LIN {X 0,Y 681.209,Z 845.598,A -85,B 0,C 180,E1 31195.432,E2 31195.432} C_VEL
LIN {X 0,Y 674.082,Z 835.285,A -85,B 0,C 180,E1 31194.524,E2 31194.524} C_VEL
LIN {X 0,Y 668.532,Z 823.271,A -85,B 0,C 180,E1 31193.574,E2 31193.574} C_VEL
LIN {X 0,Y 664.818,Z 810.324,A -85,B 0,C 180,E1 31192.643,E2 31192.643} C_VEL
LIN {X 0,Y 662.53,Z 795.041,A -85,B 0,C 180,E1 31191.638,E2 31191.638} C_VEL
LIN {X 0,Y 661.762,Z 774.741,A -85,B 0,C 180,E1 31190.407,E2 31190.407} C_VEL
LIN {X 0,Y 664.221,Z 717.539,A -85,B 0,C 180,E1 31187.123,E2 31187.123} C_VEL
LIN {X 0,Y 665.52,Z 689.484,A -85,B 0,C 180,E1 31185.472,E2 31185.472} C_VEL
LIN {X 0,Y 655.199,Z 666.535,A -85,B 0,C 180,E1 31183.253,E2 31183.253} C_VEL
LIN {X 0,Y 648.915,Z 652.729,A -85,B 0,C 180,E1 31181.851,E2 31181.851} C_VEL
LIN {X 0,Y 648.754,Z 651.857,A -85,B 0,C 180,E1 31181.745,E2 31181.745} C_VEL
LIN {X 0,Y 648.762,Z 651.857,A -85,B 0,C 180,E1 31178.737,E2 31178.737} C_VEL
LIN {X 0,Y 648.769,Z 651.859,A -85,B 0,C 180,E1 31175.632,E2 31175.632} C_VEL
LIN {X 0,Y 648.783,Z 651.97,A -85,B 0,C 180,E1 31174.365,E2 31174.365} C_VEL
LIN {X 0,Y 654.485,Z 669.215,A -85,B 0,C 180,E1 31172.597,E2 31172.597} C_VEL
LIN {X 0,Y 656.821,Z 678.025,A -85,B 0,C 180,E1 31171.733,E2 31171.733} C_VEL
LIN {X 0,Y 656.243,Z 704.05,A -85,B 0,C 180,E1 31169.628,E2 31169.628} C_VEL
LIN {X 0,Y 659.956,Z 721.319,A -85,B 0,C 180,E1 31169.192,E2 31169.192} C_VEL
LIN {X 0,Y 658.097,Z 857.869,A -85,B 0,C 180,E1 31167.489,E2 31167.489} C_VEL
LIN {X 0,Y 656.788,Z 1005.042,A -85,B 0,C 180,E1 31165.748,E2 31165.748} C_VEL
LIN {X 0,Y 656.311,Z 1027.671,A -85,B 0,C 180,E1 31165.323,E2 31165.323} C_VEL
LIN {X 0,Y 655.768,Z 1048.897,A -85,B 0,C 180,E1 31164.769,E2 31164.769} C_VEL
LIN {X 0,Y 655.075,Z 1069.242,A -85,B 0,C 180,E1 31164.083,E2 31164.083} C_VEL
LIN {X 0,Y 654.302,Z 1088.647,A -85,B 0,C 180,E1 31163.268,E2 31163.268} C_VEL
LIN {X 0,Y 653.458,Z 1107.862,A -85,B 0,C 180,E1 31162.301,E2 31162.301} C_VEL
LIN {X 0,Y 652.558,Z 1127.004,A -85,B 0,C 180,E1 31161.152,E2 31161.152} C_VEL
LIN {X 0,Y 651.651,Z 1144.284,A -85,B 0,C 180,E1 31159.916,E2 31159.916} C_VEL
LIN {X 0,Y 650.775,Z 1161.184,A -85,B 0,C 180,E1 31158.499,E2 31158.499} C_VEL
LIN {X 0,Y 650.021,Z 1176.622,A -85,B 0,C 180,E1 31156.994,E2 31156.994} C_VEL
LIN {X 0,Y 649.364,Z 1190.989,A -85,B 0,C 180,E1 31155.358,E2 31155.358} C_VEL
LIN {X 0,Y 648.862,Z 1203.128,A -85,B 0,C 180,E1 31153.728,E2 31153.728} C_VEL
LIN {X 0,Y 648.463,Z 1214.556,A -85,B 0,C 180,E1 31151.924,E2 31151.924} C_VEL
LIN {X 0,Y 648.22,Z 1224.064,A -85,B 0,C 180,E1 31150.128,E2 31150.128} C_VEL
LIN {X 0,Y 648.047,Z 1232.048,A -85,B 0,C 180,E1 31148.25,E2 31148.25} C_VEL
LIN {X 0,Y 647.962,Z 1238.272,A -85,B 0,C 180,E1 31146.379,E2 31146.379} C_VEL
LIN {X 0,Y 647.927,Z 1242.932,A -85,B 0,C 180,E1 31144.498,E2 31144.498} C_VEL
LIN {X 0,Y 647.909,Z 1245.952,A -85,B 0,C 180,E1 31142.565,E2 31142.565} C_VEL
LIN {X 0,Y 647.912,Z 1247.338,A -85,B 0,C 180,E1 31140.619,E2 31140.619} C_VEL
LIN {X 0,Y 647.903,Z 1247.184,A -85,B 0,C 180,E1 31138.762,E2 31138.762} C_VEL
LIN {X 0,Y 647.901,Z 1245.342,A -85,B 0,C 180,E1 31136.865,E2 31136.865} C_VEL
LIN {X 0,Y 647.927,Z 1241.709,A -85,B 0,C 180,E1 31134.865,E2 31134.865} C_VEL
LIN {X 0,Y 647.985,Z 1236.727,A -85,B 0,C 180,E1 31132.998,E2 31132.998} C_VEL
LIN {X 0,Y 648.081,Z 1229.943,A -85,B 0,C 180,E1 31131.125,E2 31131.125} C_VEL
LIN {X 0,Y 648.276,Z 1221.361,A -85,B 0,C 180,E1 31129.244,E2 31129.244} C_VEL
LIN {X 0,Y 648.58,Z 1211.375,A -85,B 0,C 180,E1 31127.445,E2 31127.445} C_VEL
LIN {X 0,Y 648.998,Z 1199.871,A -85,B 0,C 180,E1 31125.716,E2 31125.716} C_VEL
LIN {X 0,Y 649.525,Z 1187.153,A -85,B 0,C 180,E1 31124.096,E2 31124.096} C_VEL
LIN {X 0,Y 650.223,Z 1172.154,A -85,B 0,C 180,E1 31122.458,E2 31122.458} C_VEL
LIN {X 0,Y 651.031,Z 1156.602,A -85,B 0,C 180,E1 31120.998,E2 31120.998} C_VEL
LIN {X 0,Y 651.882,Z 1140.018,A -85,B 0,C 180,E1 31119.67,E2 31119.67} C_VEL
LIN {X 0,Y 652.795,Z 1121.9,A -85,B 0,C 180,E1 31118.432,E2 31118.432} C_VEL
LIN {X 0,Y 653.743,Z 1102.903,A -85,B 0,C 180,E1 31117.329,E2 31117.329} C_VEL
LIN {X 0,Y 654.621,Z 1083.016,A -85,B 0,C 180,E1 31116.362,E2 31116.362} C_VEL
LIN {X 0,Y 655.426,Z 1063.233,A -85,B 0,C 180,E1 31115.58,E2 31115.58} C_VEL
LIN {X 0,Y 656.167,Z 1040.826,A -85,B 0,C 180,E1 31114.87,E2 31114.87} C_VEL
LIN {X 0,Y 656.776,Z 1019.125,A -85,B 0,C 180,E1 31114.351,E2 31114.351} C_VEL
LIN {X 0,Y 657.189,Z 997.108,A -85,B 0,C 180,E1 31113.988,E2 31113.988} C_VEL
LIN {X 0,Y 657.978,Z 910.113,A -85,B 0,C 180,E1 31112.971,E2 31112.971} C_VEL
LIN {X 0,Y 657.137,Z 902.528,A -85,B 0,C 180,E1 31112.844,E2 31112.844} C_VEL
LIN {X 0,Y 651.672,Z 882.715,A -85,B 0,C 180,E1 31112.37,E2 31112.37} C_VEL
LIN {X 0,Y 651.081,Z 876.194,A -85,B 0,C 180,E1 31112.264,E2 31112.264} C_VEL
LIN {X 0,Y 652.864,Z 721.354,A -85,B 0,C 180,E1 31110.361,E2 31110.361} C_VEL
LIN {X 0,Y 648.381,Z 701.444,A -85,B 0,C 180,E1 31109.856,E2 31109.856} C_VEL
LIN {X 0,Y 649.101,Z 679.474,A -85,B 0,C 180,E1 31108.001,E2 31108.001} C_VEL
LIN {X 0,Y 642.45,Z 657.995,A -85,B 0,C 180,E1 31105.735,E2 31105.735} C_VEL
LIN {X 0,Y 640.828,Z 652.848,A -85,B 0,C 180,E1 31105.158,E2 31105.158} C_VEL
LIN {X 0,Y 640.828,Z 652.845,A -85,B 0,C 180,E1 31101.952,E2 31101.952} C_VEL
LIN {X 0,Y 640.831,Z 652.844,A -85,B 0,C 180,E1 31098.818,E2 31098.818} C_VEL
LIN {X 0,Y 640.829,Z 652.843,A -85,B 0,C 180,E1 31095.613,E2 31095.613} C_VEL
LIN {X 0,Y 640.819,Z 652.84,A -85,B 0,C 180,E1 31092.435,E2 31092.435} C_VEL
LIN {X 0,Y 640.82,Z 652.846,A -85,B 0,C 180,E1 31089.292,E2 31089.292} C_VEL
LIN {X 0,Y 640.831,Z 652.845,A -85,B 0,C 180,E1 31086.227,E2 31086.227} C_VEL
LIN {X 0,Y 640.827,Z 652.841,A -85,B 0,C 180,E1 31082.995,E2 31082.995} C_VEL
LIN {X 0,Y 640.816,Z 652.84,A -85,B 0,C 180,E1 31079.852,E2 31079.852} C_VEL
LIN {X 0,Y 640.82,Z 652.844,A -85,B 0,C 180,E1 31076.805,E2 31076.805} C_VEL
LIN {X 0,Y 640.831,Z 652.847,A -85,B 0,C 180,E1 31073.666,E2 31073.666} C_VEL
LIN {X 0,Y 640.827,Z 652.843,A -85,B 0,C 180,E1 31070.458,E2 31070.458} C_VEL
LIN {X 0,Y 640.815,Z 652.841,A -85,B 0,C 180,E1 31067.34,E2 31067.34} C_VEL
LIN {X 0,Y 640.816,Z 652.841,A -85,B 0,C 180,E1 31064.273,E2 31064.273} C_VEL
LIN {X 0,Y 640.829,Z 652.847,A -85,B 0,C 180,E1 31061.157,E2 31061.157} C_VEL
LIN {X 0,Y 640.827,Z 652.837,A -85,B 0,C 180,E1 31057.983,E2 31057.983} C_VEL
LIN {X 0,Y 640.817,Z 652.839,A -85,B 0,C 180,E1 31054.924,E2 31054.924} C_VEL
LIN {X 0,Y 640.816,Z 652.843,A -85,B 0,C 180,E1 31051.789,E2 31051.789} C_VEL
LIN {X 0,Y 640.832,Z 652.844,A -85,B 0,C 180,E1 31048.75,E2 31048.75} C_VEL
LIN {X 0,Y 640.828,Z 652.839,A -85,B 0,C 180,E1 31045.527,E2 31045.527} C_VEL
LIN {X 0,Y 640.816,Z 652.838,A -85,B 0,C 180,E1 31042.47,E2 31042.47} C_VEL
LIN {X 0,Y 640.82,Z 652.84,A -85,B 0,C 180,E1 31039.392,E2 31039.392} C_VEL
LIN {X 0,Y 640.832,Z 652.846,A -85,B 0,C 180,E1 31036.282,E2 31036.282} C_VEL
LIN {X 0,Y 640.83,Z 652.842,A -85,B 0,C 180,E1 31033.131,E2 31033.131} C_VEL
LIN {X 0,Y 640.82,Z 652.839,A -85,B 0,C 180,E1 31030.02,E2 31030.02} C_VEL
LIN {X 0,Y 640.824,Z 652.844,A -85,B 0,C 180,E1 31026.945,E2 31026.945} C_VEL
LIN {X 0,Y 640.833,Z 652.847,A -85,B 0,C 180,E1 31023.789,E2 31023.789} C_VEL
LIN {X 0,Y 640.831,Z 652.842,A -85,B 0,C 180,E1 31020.666,E2 31020.666} C_VEL
LIN {X 0,Y 640.82,Z 652.834,A -85,B 0,C 180,E1 31017.539,E2 31017.539} C_VEL
LIN {X 0,Y 640.819,Z 652.838,A -85,B 0,C 180,E1 31014.384,E2 31014.384} C_VEL
LIN {X 0,Y 640.836,Z 652.84,A -85,B 0,C 180,E1 31011.27,E2 31011.27} C_VEL
LIN {X 0,Y 640.829,Z 652.839,A -85,B 0,C 180,E1 31008.097,E2 31008.097} C_VEL
LIN {X 0,Y 640.817,Z 652.846,A -85,B 0,C 180,E1 31004.978,E2 31004.978} C_VEL
LIN {X 0,Y 640.82,Z 652.884,A -85,B 0,C 180,E1 31003.553,E2 31003.553} C_VEL
LIN {X 0,Y 650.521,Z 680.608,A -85,B 0,C 180,E1 31000.787,E2 31000.787} C_VEL
LIN {X 0,Y 651.272,Z 683.79,A -85,B 0,C 180,E1 31000.499,E2 31000.499} C_VEL
LIN {X 0,Y 649.818,Z 722.359,A -85,B 0,C 180,E1 30997.653,E2 30997.653} C_VEL
LIN {X 0,Y 648.069,Z 765.963,A -85,B 0,C 180,E1 30994.488,E2 30994.488} C_VEL
LIN {X 0,Y 646.393,Z 811.774,A -85,B 0,C 180,E1 30991.212,E2 30991.212} C_VEL
LIN {X 0,Y 644.846,Z 859.861,A -85,B 0,C 180,E1 30987.822,E2 30987.822} C_VEL
LIN {X 0,Y 643.902,Z 897.134,A -85,B 0,C 180,E1 30985.254,E2 30985.254} C_VEL
LIN {X 0,Y 644.559,Z 904.252,A -85,B 0,C 180,E1 30985.14,E2 30985.14} C_VEL
LIN {X 0,Y 643.103,Z 1040.339,A -85,B 0,C 180,E1 30983.376,E2 30983.376} C_VEL
LIN {X 0,Y 642.901,Z 1057.395,A -85,B 0,C 180,E1 30982.978,E2 30982.978} C_VEL
LIN {X 0,Y 642.615,Z 1072.675,A -85,B 0,C 180,E1 30982.451,E2 30982.451} C_VEL
LIN {X 0,Y 642.248,Z 1087.818,A -85,B 0,C 180,E1 30981.749,E2 30981.749} C_VEL
LIN {X 0,Y 641.886,Z 1101.299,A -85,B 0,C 180,E1 30980.947,E2 30980.947} C_VEL
LIN {X 0,Y 641.498,Z 1114.46,A -85,B 0,C 180,E1 30979.959,E2 30979.959} C_VEL
LIN {X 0,Y 641.17,Z 1125.58,A -85,B 0,C 180,E1 30978.928,E2 30978.928} C_VEL
LIN {X 0,Y 640.845,Z 1136.028,A -85,B 0,C 180,E1 30977.713,E2 30977.713} C_VEL
LIN {X 0,Y 640.602,Z 1144.93,A -85,B 0,C 180,E1 30976.411,E2 30976.411} C_VEL
LIN {X 0,Y 640.42,Z 1152.141,A -85,B 0,C 180,E1 30975.021,E2 30975.021} C_VEL
LIN {X 0,Y 640.328,Z 1157.431,A -85,B 0,C 180,E1 30973.638,E2 30973.638} C_VEL
LIN {X 0,Y 640.278,Z 1161.119,A -85,B 0,C 180,E1 30972.162,E2 30972.162} C_VEL
LIN {X 0,Y 640.258,Z 1163.071,A -85,B 0,C 180,E1 30970.619,E2 30970.619} C_VEL
LIN {X 0,Y 640.272,Z 1163.08,A -85,B 0,C 180,E1 30969.166,E2 30969.166} C_VEL
LIN {X 0,Y 640.325,Z 1161.258,A -85,B 0,C 180,E1 30967.627,E2 30967.627} C_VEL
LIN {X 0,Y 640.398,Z 1157.705,A -85,B 0,C 180,E1 30966.185,E2 30966.185} C_VEL
LIN {X 0,Y 640.541,Z 1152.319,A -85,B 0,C 180,E1 30964.746,E2 30964.746} C_VEL
LIN {X 0,Y 640.756,Z 1145.362,A -85,B 0,C 180,E1 30963.4,E2 30963.4} C_VEL
LIN {X 0,Y 641.066,Z 1136.322,A -85,B 0,C 180,E1 30962.056,E2 30962.056} C_VEL
LIN {X 0,Y 641.419,Z 1126.338,A -85,B 0,C 180,E1 30960.893,E2 30960.893} C_VEL
LIN {X 0,Y 641.835,Z 1114.407,A -85,B 0,C 180,E1 30959.777,E2 30959.777} C_VEL
LIN {X 0,Y 642.239,Z 1101.835,A -85,B 0,C 180,E1 30958.84,E2 30958.84} C_VEL
LIN {X 0,Y 642.653,Z 1087.565,A -85,B 0,C 180,E1 30957.994,E2 30957.994} C_VEL
LIN {X 0,Y 643.023,Z 1072.906,A -85,B 0,C 180,E1 30957.326,E2 30957.326} C_VEL
LIN {X 0,Y 643.302,Z 1057.109,A -85,B 0,C 180,E1 30956.792,E2 30956.792} C_VEL
LIN {X 0,Y 643.467,Z 1041.097,A -85,B 0,C 180,E1 30956.428,E2 30956.428} C_VEL
LIN {X 0,Y 645.88,Z 902.439,A -85,B 0,C 180,E1 30954.392,E2 30954.392} C_VEL
LIN {X 0,Y 648,Z 858.527,A -85,B 0,C 180,E1 30951.168,E2 30951.168} C_VEL
LIN {X 0,Y 650.67,Z 813.787,A -85,B 0,C 180,E1 30947.802,E2 30947.802} C_VEL
LIN {X 0,Y 653.996,Z 769.687,A -85,B 0,C 180,E1 30944.39,E2 30944.39} C_VEL
LIN {X 0,Y 657.874,Z 728.174,A -85,B 0,C 180,E1 30941.065,E2 30941.065} C_VEL
LIN {X 0,Y 660.552,Z 697.265,A -85,B 0,C 180,E1 30938.418,E2 30938.418} C_VEL
LIN {X 0,Y 655.76,Z 684.811,A -85,B 0,C 180,E1 30936.618,E2 30936.618} C_VEL
LIN {X 0,Y 651.47,Z 674.698,A -85,B 0,C 180,E1 30934.937,E2 30934.937} C_VEL
LIN {X 0,Y 647.844,Z 666.788,A -85,B 0,C 180,E1 30933.411,E2 30933.411} C_VEL
LIN {X 0,Y 646.119,Z 663.273,A -85,B 0,C 180,E1 30932.637,E2 30932.637} C_VEL
LIN {X 0,Y 643.776,Z 658.862,A -85,B 0,C 180,E1 30931.522,E2 30931.522} C_VEL
LIN {X 0,Y 643.304,Z 657.701,A -85,B 0,C 180,E1 30931.234,E2 30931.234} C_VEL
LIN {X 0,Y 641.165,Z 654.377,A -85,B 0,C 180,E1 30930.117,E2 30930.117} C_VEL
LIN {X 0,Y 640.815,Z 652.847,A -85,B 0,C 180,E1 30929.632,E2 30929.632} C_VEL
LIN {X 0,Y 640.817,Z 652.848,A -85,B 0,C 180,E1 30926.578,E2 30926.578} C_VEL
LIN {X 0,Y 640.814,Z 652.848,A -85,B 0,C 180,E1 30923.47,E2 30923.47} C_VEL
LIN {X 0,Y 640.847,Z 652.979,A -85,B 0,C 180,E1 30921.097,E2 30921.097} C_VEL
LIN {X 0,Y 642.181,Z 656.406,A -85,B 0,C 180,E1 30920.213,E2 30920.213} C_VEL
LIN {X 0,Y 643.755,Z 658.201,A -85,B 0,C 180,E1 30919.632,E2 30919.632} C_VEL
LIN {X 0,Y 645.497,Z 662.058,A -85,B 0,C 180,E1 30918.827,E2 30918.827} C_VEL
LIN {X 0,Y 646.606,Z 663.902,A -85,B 0,C 180,E1 30918.441,E2 30918.441} C_VEL
LIN {X 0,Y 649.083,Z 668.897,A -85,B 0,C 180,E1 30917.549,E2 30917.549} C_VEL
LIN {X 0,Y 652.65,Z 676.198,A -85,B 0,C 180,E1 30916.415,E2 30916.415} C_VEL
LIN {X 0,Y 657.722,Z 688.151,A -85,B 0,C 180,E1 30914.893,E2 30914.893} C_VEL
LIN {X 0,Y 658.832,Z 691.207,A -85,B 0,C 180,E1 30914.557,E2 30914.557} C_VEL
LIN {X 0,Y 654.691,Z 733.352,A -85,B 0,C 180,E1 30911.945,E2 30911.945} C_VEL
LIN {X 0,Y 652.167,Z 775.541,A -85,B 0,C 180,E1 30909.449,E2 30909.449} C_VEL
LIN {X 0,Y 653.059,Z 796.061,A -85,B 0,C 180,E1 30908.174,E2 30908.174} C_VEL
LIN {X 0,Y 655.531,Z 811.396,A -85,B 0,C 180,E1 30907.156,E2 30907.156} C_VEL
LIN {X 0,Y 659.426,Z 824.494,A -85,B 0,C 180,E1 30906.227,E2 30906.227} C_VEL
LIN {X 0,Y 665.197,Z 836.86,A -85,B 0,C 180,E1 30905.292,E2 30905.292} C_VEL
LIN {X 0,Y 672.623,Z 847.758,A -85,B 0,C 180,E1 30904.407,E2 30904.407} C_VEL
LIN {X 0,Y 681.659,Z 857.265,A -85,B 0,C 180,E1 30903.574,E2 30903.574} C_VEL
LIN {X 0,Y 691.482,Z 864.868,A -85,B 0,C 180,E1 30902.845,E2 30902.845} C_VEL
LIN {X 0,Y 702.753,Z 871.277,A -85,B 0,C 180,E1 30902.158,E2 30902.158} C_VEL
LIN {X 0,Y 715.436,Z 876.288,A -85,B 0,C 180,E1 30901.511,E2 30901.511} C_VEL
LIN {X 0,Y 720.879,Z 877.314,A -85,B 0,C 180,E1 30901.151,E2 30901.151} C_VEL
LIN {X 0,Y 724.061,Z 877.311,A -85,B 0,C 180,E1 30900.847,E2 30900.847} C_VEL
LIN {X 0,Y 720.157,Z 886.663,A -85,B 0,C 180,E1 30900.632,E2 30900.632} C_VEL
LIN {X 0,Y 710.62,Z 902.495,A -85,B 0,C 180,E1 30900.397,E2 30900.397} C_VEL
LIN {X 0,Y 697.384,Z 921.767,A -85,B 0,C 180,E1 30899.929,E2 30899.929} C_VEL
LIN {X 0,Y 679.73,Z 948.078,A -85,B 0,C 180,E1 30899.184,E2 30899.184} C_VEL
LIN {X 0,Y 670.449,Z 964.538,A -85,B 0,C 180,E1 30898.649,E2 30898.649} C_VEL
LIN {X 0,Y 664.344,Z 978.497,A -85,B 0,C 180,E1 30898.136,E2 30898.136} C_VEL
LIN {X 0,Y 662.043,Z 984.008,A -85,B 0,C 180,E1 30897.928,E2 30897.928} C_VEL
LIN {X 0,Y 656.266,Z 997.296,A -85,B 0,C 180,E1 30897.428,E2 30897.428} C_VEL
LIN {X 0,Y 650.15,Z 1017.526,A -85,B 0,C 180,E1 30896.584,E2 30896.584} C_VEL
LIN {X 0,Y 649.41,Z 1021.143,A -85,B 0,C 180,E1 30896.453,E2 30896.453} C_VEL
LIN {X 0,Y 648.837,Z 1062.962,A -85,B 0,C 180,E1 30895.95,E2 30895.95} C_VEL
LIN {X 0,Y 648.281,Z 1086.804,A -85,B 0,C 180,E1 30895.491,E2 30895.491} C_VEL
LIN {X 0,Y 647.655,Z 1109.654,A -85,B 0,C 180,E1 30894.877,E2 30894.877} C_VEL
LIN {X 0,Y 646.894,Z 1131.523,A -85,B 0,C 180,E1 30894.115,E2 30894.115} C_VEL
LIN {X 0,Y 646.063,Z 1153.311,A -85,B 0,C 180,E1 30893.173,E2 30893.173} C_VEL
LIN {X 0,Y 645.207,Z 1173.52,A -85,B 0,C 180,E1 30892.12,E2 30892.12} C_VEL
LIN {X 0,Y 644.365,Z 1192.384,A -85,B 0,C 180,E1 30890.956,E2 30890.956} C_VEL
LIN {X 0,Y 643.526,Z 1209.876,A -85,B 0,C 180,E1 30889.68,E2 30889.68} C_VEL
LIN {X 0,Y 642.771,Z 1226.068,A -85,B 0,C 180,E1 30888.313,E2 30888.313} C_VEL
LIN {X 0,Y 642.061,Z 1239.527,A -85,B 0,C 180,E1 30886.929,E2 30886.929} C_VEL
LIN {X 0,Y 641.481,Z 1251.253,A -85,B 0,C 180,E1 30885.55,E2 30885.55} C_VEL
LIN {X 0,Y 640.968,Z 1262.832,A -85,B 0,C 180,E1 30883.991,E2 30883.991} C_VEL
LIN {X 0,Y 640.52,Z 1274.803,A -85,B 0,C 180,E1 30882.073,E2 30882.073} C_VEL
LIN {X 0,Y 640.251,Z 1283.342,A -85,B 0,C 180,E1 30880.436,E2 30880.436} C_VEL
LIN {X 0,Y 640.081,Z 1290.854,A -85,B 0,C 180,E1 30878.714,E2 30878.714} C_VEL
LIN {X 0,Y 639.963,Z 1297.62,A -85,B 0,C 180,E1 30876.728,E2 30876.728} C_VEL
LIN {X 0,Y 639.927,Z 1301.986,A -85,B 0,C 180,E1 30875.019,E2 30875.019} C_VEL
LIN {X 0,Y 639.919,Z 1305.213,A -85,B 0,C 180,E1 30873.223,E2 30873.223} C_VEL
LIN {X 0,Y 639.914,Z 1307.192,A -85,B 0,C 180,E1 30871.073,E2 30871.073} C_VEL
LIN {X 0,Y 639.904,Z 1307.328,A -85,B 0,C 180,E1 30869.372,E2 30869.372} C_VEL
LIN {X 0,Y 639.905,Z 1306.259,A -85,B 0,C 180,E1 30867.67,E2 30867.67} C_VEL
LIN {X 0,Y 639.923,Z 1303.51,A -85,B 0,C 180,E1 30865.698,E2 30865.698} C_VEL
LIN {X 0,Y 639.952,Z 1299.128,A -85,B 0,C 180,E1 30863.81,E2 30863.81} C_VEL
LIN {X 0,Y 640.019,Z 1294.119,A -85,B 0,C 180,E1 30862.187,E2 30862.187} C_VEL
LIN {X 0,Y 640.162,Z 1287.481,A -85,B 0,C 180,E1 30860.469,E2 30860.469} C_VEL
LIN {X 0,Y 640.42,Z 1277.822,A -85,B 0,C 180,E1 30858.471,E2 30858.471} C_VEL
LIN {X 0,Y 640.728,Z 1268.768,A -85,B 0,C 180,E1 30856.921,E2 30856.921} C_VEL
LIN {X 0,Y 641.138,Z 1258.901,A -85,B 0,C 180,E1 30855.457,E2 30855.457} C_VEL
LIN {X 0,Y 641.747,Z 1246.072,A -85,B 0,C 180,E1 30853.805,E2 30853.805} C_VEL
LIN {X 0,Y 642.465,Z 1231.649,A -85,B 0,C 180,E1 30852.238,E2 30852.238} C_VEL
LIN {X 0,Y 643.038,Z 1220.295,A -85,B 0,C 180,E1 30851.176,E2 30851.176} C_VEL
LIN {X 0,Y 643.729,Z 1206.008,A -85,B 0,C 180,E1 30850.008,E2 30850.008} C_VEL
LIN {X 0,Y 644.577,Z 1189.105,A -85,B 0,C 180,E1 30848.796,E2 30848.796} C_VEL
LIN {X 0,Y 645.498,Z 1169.439,A -85,B 0,C 180,E1 30847.6,E2 30847.6} C_VEL
LIN {X 0,Y 646.44,Z 1148.388,A -85,B 0,C 180,E1 30846.525,E2 30846.525} C_VEL
LIN {X 0,Y 647.307,Z 1127.423,A -85,B 0,C 180,E1 30845.641,E2 30845.641} C_VEL
LIN {X 0,Y 648.102,Z 1105.683,A -85,B 0,C 180,E1 30844.908,E2 30844.908} C_VEL
LIN {X 0,Y 648.775,Z 1083.009,A -85,B 0,C 180,E1 30844.321,E2 30844.321} C_VEL
LIN {X 0,Y 649.317,Z 1060.66,A -85,B 0,C 180,E1 30843.904,E2 30843.904} C_VEL
LIN {X 0,Y 649.898,Z 1021.34,A -85,B 0,C 180,E1 30843.427,E2 30843.427} C_VEL
LIN {X 0,Y 653.512,Z 1008.382,A -85,B 0,C 180,E1 30842.873,E2 30842.873} C_VEL
LIN {X 0,Y 658.239,Z 994.241,A -85,B 0,C 180,E1 30842.3,E2 30842.3} C_VEL
LIN {X 0,Y 664.396,Z 980.423,A -85,B 0,C 180,E1 30841.799,E2 30841.799} C_VEL
LIN {X 0,Y 669.874,Z 967.309,A -85,B 0,C 180,E1 30841.321,E2 30841.321} C_VEL
LIN {X 0,Y 678.652,Z 950.97,A -85,B 0,C 180,E1 30840.811,E2 30840.811} C_VEL
LIN {X 0,Y 693.309,Z 928.11,A -85,B 0,C 180,E1 30840.203,E2 30840.203} C_VEL
LIN {X 0,Y 712.087,Z 900.21,A -85,B 0,C 180,E1 30839.561,E2 30839.561} C_VEL
LIN {X 0,Y 720.725,Z 885.47,A -85,B 0,C 180,E1 30839.346,E2 30839.346} C_VEL
LIN {X 0,Y 724.073,Z 877.281,A -85,B 0,C 180,E1 30839.152,E2 30839.152} C_VEL
LIN {X 0,Y 719.403,Z 877.155,A -85,B 0,C 180,E1 30838.736,E2 30838.736} C_VEL
LIN {X 0,Y 713.768,Z 875.787,A -85,B 0,C 180,E1 30838.4,E2 30838.4} C_VEL
LIN {X 0,Y 701.67,Z 871.121,A -85,B 0,C 180,E1 30837.676,E2 30837.676} C_VEL
LIN {X 0,Y 691.019,Z 865.082,A -85,B 0,C 180,E1 30836.909,E2 30836.909} C_VEL
LIN {X 0,Y 681.773,Z 857.782,A -85,B 0,C 180,E1 30836.109,E2 30836.109} C_VEL
LIN {X 0,Y 673.653,Z 848.946,A -85,B 0,C 180,E1 30835.252,E2 30835.252} C_VEL
LIN {X 0,Y 666.592,Z 838.079,A -85,B 0,C 180,E1 30834.302,E2 30834.302} C_VEL
LIN {X 0,Y 661.173,Z 825.61,A -85,B 0,C 180,E1 30833.318,E2 30833.318} C_VEL
LIN {X 0,Y 657.433,Z 811.523,A -85,B 0,C 180,E1 30832.308,E2 30832.308} C_VEL
LIN {X 0,Y 655.376,Z 795.861,A -85,B 0,C 180,E1 30831.278,E2 30831.278} C_VEL
LIN {X 0,Y 654.815,Z 775.606,A -85,B 0,C 180,E1 30830.045,E2 30830.045} C_VEL
LIN {X 0,Y 657.442,Z 719.808,A -85,B 0,C 180,E1 30826.811,E2 30826.811} C_VEL
LIN {X 0,Y 658.829,Z 693.191,A -85,B 0,C 180,E1 30825.234,E2 30825.234} C_VEL
LIN {X 0,Y 647.655,Z 668.207,A -85,B 0,C 180,E1 30822.789,E2 30822.789} C_VEL
LIN {X 0,Y 641.688,Z 655.612,A -85,B 0,C 180,E1 30821.471,E2 30821.471} C_VEL
LIN {X 0,Y 640.829,Z 652.848,A -85,B 0,C 180,E1 30821.182,E2 30821.182} C_VEL
LIN {X 0,Y 640.832,Z 652.847,A -85,B 0,C 180,E1 30818.005,E2 30818.005} C_VEL
LIN {X 0,Y 640.861,Z 653.038,A -85,B 0,C 180,E1 30814.846,E2 30814.846} C_VEL
LIN {X 0,Y 646.617,Z 669.593,A -85,B 0,C 180,E1 30813.084,E2 30813.084} C_VEL
LIN {X 0,Y 649.738,Z 680.661,A -85,B 0,C 180,E1 30811.964,E2 30811.964} C_VEL
LIN {X 0,Y 649.191,Z 704.841,A -85,B 0,C 180,E1 30810.004,E2 30810.004} C_VEL
LIN {X 0,Y 653.002,Z 722.678,A -85,B 0,C 180,E1 30809.526,E2 30809.526} C_VEL
LIN {X 0,Y 650.797,Z 859.006,A -85,B 0,C 180,E1 30807.766,E2 30807.766} C_VEL
LIN {X 0,Y 649.316,Z 1005.981,A -85,B 0,C 180,E1 30805.99,E2 30805.99} C_VEL
LIN {X 0,Y 648.819,Z 1028.459,A -85,B 0,C 180,E1 30805.561,E2 30805.561} C_VEL
LIN {X 0,Y 648.22,Z 1050.332,A -85,B 0,C 180,E1 30804.978,E2 30804.978} C_VEL
LIN {X 0,Y 647.477,Z 1071.362,A -85,B 0,C 180,E1 30804.254,E2 30804.254} C_VEL
LIN {X 0,Y 646.61,Z 1091.799,A -85,B 0,C 180,E1 30803.368,E2 30803.368} C_VEL
LIN {X 0,Y 645.678,Z 1111.353,A -85,B 0,C 180,E1 30802.345,E2 30802.345} C_VEL
LIN {X 0,Y 644.8,Z 1128.969,A -85,B 0,C 180,E1 30801.255,E2 30801.255} C_VEL
LIN {X 0,Y 643.884,Z 1145.8,A -85,B 0,C 180,E1 30800.03,E2 30800.03} C_VEL
LIN {X 0,Y 643.019,Z 1161.653,A -85,B 0,C 180,E1 30798.683,E2 30798.683} C_VEL
LIN {X 0,Y 642.227,Z 1176.625,A -85,B 0,C 180,E1 30797.206,E2 30797.206} C_VEL
LIN {X 0,Y 641.508,Z 1190.991,A -85,B 0,C 180,E1 30795.551,E2 30795.551} C_VEL
LIN {X 0,Y 640.956,Z 1203.13,A -85,B 0,C 180,E1 30793.901,E2 30793.901} C_VEL
LIN {X 0,Y 640.52,Z 1214.557,A -85,B 0,C 180,E1 30792.074,E2 30792.074} C_VEL
LIN {X 0,Y 640.252,Z 1224.067,A -85,B 0,C 180,E1 30790.255,E2 30790.255} C_VEL
LIN {X 0,Y 640.056,Z 1232.05,A -85,B 0,C 180,E1 30788.354,E2 30788.354} C_VEL
LIN {X 0,Y 639.964,Z 1238.342,A -85,B 0,C 180,E1 30786.435,E2 30786.435} C_VEL
LIN {X 0,Y 639.927,Z 1242.984,A -85,B 0,C 180,E1 30784.525,E2 30784.525} C_VEL
LIN {X 0,Y 639.91,Z 1245.952,A -85,B 0,C 180,E1 30782.597,E2 30782.597} C_VEL
LIN {X 0,Y 639.912,Z 1247.338,A -85,B 0,C 180,E1 30780.627,E2 30780.627} C_VEL
LIN {X 0,Y 639.903,Z 1247.184,A -85,B 0,C 180,E1 30778.746,E2 30778.746} C_VEL
LIN {X 0,Y 639.901,Z 1245.367,A -85,B 0,C 180,E1 30776.847,E2 30776.847} C_VEL
LIN {X 0,Y 639.93,Z 1241.708,A -85,B 0,C 180,E1 30774.8,E2 30774.8} C_VEL
LIN {X 0,Y 639.993,Z 1236.725,A -85,B 0,C 180,E1 30772.91,E2 30772.91} C_VEL
LIN {X 0,Y 640.103,Z 1229.941,A -85,B 0,C 180,E1 30771.013,E2 30771.013} C_VEL
LIN {X 0,Y 640.317,Z 1221.357,A -85,B 0,C 180,E1 30769.109,E2 30769.109} C_VEL
LIN {X 0,Y 640.648,Z 1211.348,A -85,B 0,C 180,E1 30767.284,E2 30767.284} C_VEL
LIN {X 0,Y 641.103,Z 1199.957,A -85,B 0,C 180,E1 30765.549,E2 30765.549} C_VEL
LIN {X 0,Y 641.686,Z 1187.145,A -85,B 0,C 180,E1 30763.897,E2 30763.897} C_VEL
LIN {X 0,Y 642.445,Z 1172.146,A -85,B 0,C 180,E1 30762.239,E2 30762.239} C_VEL
LIN {X 0,Y 643.315,Z 1156.535,A -85,B 0,C 180,E1 30760.761,E2 30760.761} C_VEL
LIN {X 0,Y 644.234,Z 1139.851,A -85,B 0,C 180,E1 30759.418,E2 30759.418} C_VEL
LIN {X 0,Y 645.202,Z 1121.709,A -85,B 0,C 180,E1 30758.171,E2 30758.171} C_VEL
LIN {X 0,Y 646.216,Z 1102.486,A -85,B 0,C 180,E1 30757.05,E2 30757.05} C_VEL
LIN {X 0,Y 647.149,Z 1082.872,A -85,B 0,C 180,E1 30756.09,E2 30756.09} C_VEL
LIN {X 0,Y 648.022,Z 1062.526,A -85,B 0,C 180,E1 30755.282,E2 30755.282} C_VEL
LIN {X 0,Y 648.786,Z 1040.647,A -85,B 0,C 180,E1 30754.588,E2 30754.588} C_VEL
LIN {X 0,Y 649.426,Z 1018.944,A -85,B 0,C 180,E1 30754.067,E2 30754.067} C_VEL
LIN {X 0,Y 649.868,Z 997.018,A -85,B 0,C 180,E1 30753.702,E2 30753.702} C_VEL
LIN {X 0,Y 651.081,Z 876.194,A -85,B 0,C 180,E1 30752.264,E2 30752.264} C_VEL
LIN {X 0,Y 650.293,Z 868.612,A -85,B 0,C 180,E1 30752.135,E2 30752.135} C_VEL
LIN {X 0,Y 644.932,Z 848.819,A -85,B 0,C 180,E1 30751.641,E2 30751.641} C_VEL
LIN {X 0,Y 644.334,Z 842.302,A -85,B 0,C 180,E1 30751.531,E2 30751.531} C_VEL
LIN {X 0,Y 645.843,Z 722.596,A -85,B 0,C 180,E1 30750.022,E2 30750.022} C_VEL
LIN {X 0,Y 641.129,Z 701.54,A -85,B 0,C 180,E1 30749.471,E2 30749.471} C_VEL
LIN {X 0,Y 641.677,Z 681.932,A -85,B 0,C 180,E1 30747.794,E2 30747.794} C_VEL
LIN {X 0,Y 635.199,Z 661.095,A -85,B 0,C 180,E1 30745.574,E2 30745.574} C_VEL
LIN {X 0,Y 632.877,Z 653.837,A -85,B 0,C 180,E1 30744.768,E2 30744.768} C_VEL
LIN {X 0,Y 632.878,Z 653.836,A -85,B 0,C 180,E1 30741.733,E2 30741.733} C_VEL
LIN {X 0,Y 632.889,Z 653.833,A -85,B 0,C 180,E1 30738.63,E2 30738.63} C_VEL
LIN {X 0,Y 632.888,Z 653.834,A -85,B 0,C 180,E1 30735.442,E2 30735.442} C_VEL
LIN {X 0,Y 632.875,Z 653.83,A -85,B 0,C 180,E1 30732.303,E2 30732.303} C_VEL
LIN {X 0,Y 632.877,Z 653.835,A -85,B 0,C 180,E1 30729.196,E2 30729.196} C_VEL
LIN {X 0,Y 632.892,Z 653.836,A -85,B 0,C 180,E1 30726.108,E2 30726.108} C_VEL
LIN {X 0,Y 632.888,Z 653.831,A -85,B 0,C 180,E1 30722.922,E2 30722.922} C_VEL
LIN {X 0,Y 632.877,Z 653.829,A -85,B 0,C 180,E1 30719.845,E2 30719.845} C_VEL
LIN {X 0,Y 632.879,Z 653.832,A -85,B 0,C 180,E1 30716.762,E2 30716.762} C_VEL
LIN {X 0,Y 632.892,Z 653.836,A -85,B 0,C 180,E1 30713.66,E2 30713.66} C_VEL
LIN {X 0,Y 632.888,Z 653.832,A -85,B 0,C 180,E1 30710.437,E2 30710.437} C_VEL
LIN {X 0,Y 632.878,Z 653.83,A -85,B 0,C 180,E1 30707.375,E2 30707.375} C_VEL
LIN {X 0,Y 632.877,Z 653.829,A -85,B 0,C 180,E1 30704.27,E2 30704.27} C_VEL
LIN {X 0,Y 632.891,Z 653.836,A -85,B 0,C 180,E1 30701.155,E2 30701.155} C_VEL
LIN {X 0,Y 632.888,Z 653.826,A -85,B 0,C 180,E1 30697.993,E2 30697.993} C_VEL
LIN {X 0,Y 632.877,Z 653.829,A -85,B 0,C 180,E1 30694.895,E2 30694.895} C_VEL
LIN {X 0,Y 632.878,Z 653.832,A -85,B 0,C 180,E1 30691.812,E2 30691.812} C_VEL
LIN {X 0,Y 632.894,Z 653.833,A -85,B 0,C 180,E1 30688.734,E2 30688.734} C_VEL
LIN {X 0,Y 632.889,Z 653.828,A -85,B 0,C 180,E1 30685.496,E2 30685.496} C_VEL
LIN {X 0,Y 632.874,Z 653.827,A -85,B 0,C 180,E1 30682.375,E2 30682.375} C_VEL
LIN {X 0,Y 632.874,Z 653.828,A -85,B 0,C 180,E1 30679.257,E2 30679.257} C_VEL
LIN {X 0,Y 632.893,Z 653.833,A -85,B 0,C 180,E1 30676.2,E2 30676.2} C_VEL
LIN {X 0,Y 632.89,Z 653.833,A -85,B 0,C 180,E1 30673.007,E2 30673.007} C_VEL
LIN {X 0,Y 632.874,Z 653.829,A -85,B 0,C 180,E1 30669.855,E2 30669.855} C_VEL
LIN {X 0,Y 632.875,Z 653.833,A -85,B 0,C 180,E1 30666.737,E2 30666.737} C_VEL
LIN {X 0,Y 632.891,Z 653.834,A -85,B 0,C 180,E1 30663.611,E2 30663.611} C_VEL
LIN {X 0,Y 632.89,Z 653.833,A -85,B 0,C 180,E1 30660.469,E2 30660.469} C_VEL
LIN {X 0,Y 632.875,Z 653.824,A -85,B 0,C 180,E1 30657.363,E2 30657.363} C_VEL
LIN {X 0,Y 632.876,Z 653.826,A -85,B 0,C 180,E1 30654.3,E2 30654.3} C_VEL
LIN {X 0,Y 632.897,Z 653.829,A -85,B 0,C 180,E1 30651.274,E2 30651.274} C_VEL
LIN {X 0,Y 632.89,Z 653.827,A -85,B 0,C 180,E1 30648.067,E2 30648.067} C_VEL
LIN {X 0,Y 632.877,Z 653.835,A -85,B 0,C 180,E1 30644.929,E2 30644.929} C_VEL
LIN {X 0,Y 632.895,Z 653.934,A -85,B 0,C 180,E1 30643.979,E2 30643.979} C_VEL
LIN {X 0,Y 642.368,Z 680.772,A -85,B 0,C 180,E1 30641.254,E2 30641.254} C_VEL
LIN {X 0,Y 644.069,Z 686.626,A -85,B 0,C 180,E1 30640.695,E2 30640.695} C_VEL
LIN {X 0,Y 642.491,Z 725.275,A -85,B 0,C 180,E1 30637.819,E2 30637.819} C_VEL
LIN {X 0,Y 640.685,Z 768.41,A -85,B 0,C 180,E1 30634.671,E2 30634.671} C_VEL
LIN {X 0,Y 638.927,Z 813.648,A -85,B 0,C 180,E1 30631.408,E2 30631.408} C_VEL
LIN {X 0,Y 637.26,Z 862.229,A -85,B 0,C 180,E1 30627.953,E2 30627.953} C_VEL
LIN {X 0,Y 636.301,Z 897.732,A -85,B 0,C 180,E1 30625.487,E2 30625.487} C_VEL
LIN {X 0,Y 636.992,Z 905.112,A -85,B 0,C 180,E1 30625.365,E2 30625.365} C_VEL
LIN {X 0,Y 635.378,Z 1041.243,A -85,B 0,C 180,E1 30623.551,E2 30623.551} C_VEL
LIN {X 0,Y 635.166,Z 1058.163,A -85,B 0,C 180,E1 30623.148,E2 30623.148} C_VEL
LIN {X 0,Y 634.854,Z 1073.763,A -85,B 0,C 180,E1 30622.6,E2 30622.6} C_VEL
LIN {X 0,Y 634.459,Z 1089.03,A -85,B 0,C 180,E1 30621.879,E2 30621.879} C_VEL
LIN {X 0,Y 634.075,Z 1102.331,A -85,B 0,C 180,E1 30621.072,E2 30621.072} C_VEL
LIN {X 0,Y 633.642,Z 1116.015,A -85,B 0,C 180,E1 30620.025,E2 30620.025} C_VEL
LIN {X 0,Y 633.286,Z 1127.126,A -85,B 0,C 180,E1 30618.965,E2 30618.965} C_VEL
LIN {X 0,Y 632.939,Z 1137.568,A -85,B 0,C 180,E1 30617.72,E2 30617.72} C_VEL
LIN {X 0,Y 632.679,Z 1146.269,A -85,B 0,C 180,E1 30616.409,E2 30616.409} C_VEL
LIN {X 0,Y 632.489,Z 1153.353,A -85,B 0,C 180,E1 30615.01,E2 30615.01} C_VEL
LIN {X 0,Y 632.392,Z 1158.522,A -85,B 0,C 180,E1 30613.626,E2 30613.626} C_VEL
LIN {X 0,Y 632.335,Z 1162.131,A -85,B 0,C 180,E1 30612.14,E2 30612.14} C_VEL
LIN {X 0,Y 632.315,Z 1163.988,A -85,B 0,C 180,E1 30610.662,E2 30610.662} C_VEL
LIN {X 0,Y 632.33,Z 1164.067,A -85,B 0,C 180,E1 30609.19,E2 30609.19} C_VEL
LIN {X 0,Y 632.391,Z 1162.301,A -85,B 0,C 180,E1 30607.632,E2 30607.632} C_VEL
LIN {X 0,Y 632.476,Z 1158.821,A -85,B 0,C 180,E1 30606.171,E2 30606.171} C_VEL
LIN {X 0,Y 632.633,Z 1153.498,A -85,B 0,C 180,E1 30604.714,E2 30604.714} C_VEL
LIN {X 0,Y 632.872,Z 1146.628,A -85,B 0,C 180,E1 30603.351,E2 30603.351} C_VEL
LIN {X 0,Y 633.208,Z 1137.669,A -85,B 0,C 180,E1 30601.991,E2 30601.991} C_VEL
LIN {X 0,Y 633.591,Z 1127.807,A -85,B 0,C 180,E1 30600.814,E2 30600.814} C_VEL
LIN {X 0,Y 634.036,Z 1115.999,A -85,B 0,C 180,E1 30599.684,E2 30599.684} C_VEL
LIN {X 0,Y 634.478,Z 1103.644,A -85,B 0,C 180,E1 30598.736,E2 30598.736} C_VEL
LIN {X 0,Y 634.915,Z 1089.624,A -85,B 0,C 180,E1 30597.879,E2 30597.879} C_VEL
LIN {X 0,Y 635.329,Z 1075.481,A -85,B 0,C 180,E1 30597.204,E2 30597.204} C_VEL
LIN {X 0,Y 635.634,Z 1059.544,A -85,B 0,C 180,E1 30596.641,E2 30596.641} C_VEL
LIN {X 0,Y 635.832,Z 1043.549,A -85,B 0,C 180,E1 30596.25,E2 30596.25} C_VEL
LIN {X 0,Y 638.592,Z 903.724,A -85,B 0,C 180,E1 30594.113,E2 30594.113} C_VEL
LIN {X 0,Y 640.89,Z 859.699,A -85,B 0,C 180,E1 30590.843,E2 30590.843} C_VEL
LIN {X 0,Y 643.769,Z 815.073,A -85,B 0,C 180,E1 30587.441,E2 30587.441} C_VEL
LIN {X 0,Y 647.321,Z 771.75,A -85,B 0,C 180,E1 30584.041,E2 30584.041} C_VEL
LIN {X 0,Y 651.422,Z 730.897,A -85,B 0,C 180,E1 30580.725,E2 30580.725} C_VEL
LIN {X 0,Y 654.217,Z 701.38,A -85,B 0,C 180,E1 30578.151,E2 30578.151} C_VEL
LIN {X 0,Y 649.25,Z 688.122,A -85,B 0,C 180,E1 30576.172,E2 30576.172} C_VEL
LIN {X 0,Y 644.531,Z 676.958,A -85,B 0,C 180,E1 30574.2,E2 30574.2} C_VEL
LIN {X 0,Y 641.753,Z 671.469,A -85,B 0,C 180,E1 30573.021,E2 30573.021} C_VEL
LIN {X 0,Y 640.285,Z 668.158,A -85,B 0,C 180,E1 30572.266,E2 30572.266} C_VEL
LIN {X 0,Y 638.593,Z 664.72,A -85,B 0,C 180,E1 30571.372,E2 30571.372} C_VEL
LIN {X 0,Y 637.71,Z 663.298,A -85,B 0,C 180,E1 30570.918,E2 30570.918} C_VEL
LIN {X 0,Y 635.923,Z 659.39,A -85,B 0,C 180,E1 30569.676,E2 30569.676} C_VEL
LIN {X 0,Y 633.291,Z 655.558,A -85,B 0,C 180,E1 30567.532,E2 30567.532} C_VEL
LIN {X 0,Y 632.888,Z 653.836,A -85,B 0,C 180,E1 30566.103,E2 30566.103} C_VEL
LIN {X 0,Y 632.924,Z 654.095,A -85,B 0,C 180,E1 30564.23,E2 30564.23} C_VEL
LIN {X 0,Y 634.036,Z 657.091,A -85,B 0,C 180,E1 30562.388,E2 30562.388} C_VEL
LIN {X 0,Y 636.14,Z 659.562,A -85,B 0,C 180,E1 30561.159,E2 30561.159} C_VEL
LIN {X 0,Y 637.618,Z 663.036,A -85,B 0,C 180,E1 30560.207,E2 30560.207} C_VEL
LIN {X 0,Y 638.838,Z 664.574,A -85,B 0,C 180,E1 30559.728,E2 30559.728} C_VEL
LIN {X 0,Y 640.873,Z 668.658,A -85,B 0,C 180,E1 30558.821,E2 30558.821} C_VEL
LIN {X 0,Y 643.983,Z 675.08,A -85,B 0,C 180,E1 30557.634,E2 30557.634} C_VEL
LIN {X 0,Y 647.435,Z 682.518,A -85,B 0,C 180,E1 30556.465,E2 30556.465} C_VEL
LIN {X 0,Y 651.923,Z 693.301,A -85,B 0,C 180,E1 30555.065,E2 30555.065} C_VEL
LIN {X 0,Y 652.46,Z 695.654,A -85,B 0,C 180,E1 30554.823,E2 30554.823} C_VEL
LIN {X 0,Y 647.951,Z 737.834,A -85,B 0,C 180,E1 30552.163,E2 30552.163} C_VEL
LIN {X 0,Y 645.277,Z 778.02,A -85,B 0,C 180,E1 30549.735,E2 30549.735} C_VEL
LIN {X 0,Y 646.01,Z 798.303,A -85,B 0,C 180,E1 30548.447,E2 30548.447} C_VEL
LIN {X 0,Y 648.312,Z 813.638,A -85,B 0,C 180,E1 30547.412,E2 30547.412} C_VEL
LIN {X 0,Y 652.281,Z 827.583,A -85,B 0,C 180,E1 30546.411,E2 30546.411} C_VEL
LIN {X 0,Y 658.185,Z 840.595,A -85,B 0,C 180,E1 30545.409,E2 30545.409} C_VEL
LIN {X 0,Y 665.481,Z 851.613,A -85,B 0,C 180,E1 30544.501,E2 30544.501} C_VEL
LIN {X 0,Y 674.012,Z 861.011,A -85,B 0,C 180,E1 30543.67,E2 30543.67} C_VEL
LIN {X 0,Y 683.687,Z 869.014,A -85,B 0,C 180,E1 30542.915,E2 30542.915} C_VEL
LIN {X 0,Y 694.798,Z 875.887,A -85,B 0,C 180,E1 30542.199,E2 30542.199} C_VEL
LIN {X 0,Y 707.352,Z 881.469,A -85,B 0,C 180,E1 30541.528,E2 30541.528} C_VEL
LIN {X 0,Y 715.316,Z 884.147,A -85,B 0,C 180,E1 30541.12,E2 30541.12} C_VEL
LIN {X 0,Y 698.984,Z 907.569,A -85,B 0,C 180,E1 30540.553,E2 30540.553} C_VEL
LIN {X 0,Y 674.952,Z 942.623,A -85,B 0,C 180,E1 30539.588,E2 30539.588} C_VEL
LIN {X 0,Y 664.645,Z 960.325,A -85,B 0,C 180,E1 30539.022,E2 30539.022} C_VEL
LIN {X 0,Y 657.997,Z 974.762,A -85,B 0,C 180,E1 30538.498,E2 30538.498} C_VEL
LIN {X 0,Y 655.226,Z 981.685,A -85,B 0,C 180,E1 30538.232,E2 30538.232} C_VEL
LIN {X 0,Y 649.203,Z 995.335,A -85,B 0,C 180,E1 30537.717,E2 30537.717} C_VEL
LIN {X 0,Y 642.641,Z 1016.703,A -85,B 0,C 180,E1 30536.82,E2 30536.82} C_VEL
LIN {X 0,Y 642.258,Z 1019.206,A -85,B 0,C 180,E1 30536.76,E2 30536.76} C_VEL
LIN {X 0,Y 641.745,Z 1039.661,A -85,B 0,C 180,E1 30536.528,E2 30536.528} C_VEL
LIN {X 0,Y 641.324,Z 1068.043,A -85,B 0,C 180,E1 30536.14,E2 30536.14} C_VEL
LIN {X 0,Y 640.725,Z 1090.613,A -85,B 0,C 180,E1 30535.66,E2 30535.66} C_VEL
LIN {X 0,Y 639.967,Z 1112.73,A -85,B 0,C 180,E1 30535.014,E2 30535.014} C_VEL
LIN {X 0,Y 639.082,Z 1134.545,A -85,B 0,C 180,E1 30534.196,E2 30534.196} C_VEL
LIN {X 0,Y 638.096,Z 1156.974,A -85,B 0,C 180,E1 30533.159,E2 30533.159} C_VEL
LIN {X 0,Y 637.204,Z 1176.757,A -85,B 0,C 180,E1 30532.073,E2 30532.073} C_VEL
LIN {X 0,Y 636.276,Z 1196.341,A -85,B 0,C 180,E1 30530.801,E2 30530.801} C_VEL
LIN {X 0,Y 635.327,Z 1215.225,A -85,B 0,C 180,E1 30529.345,E2 30529.345} C_VEL
LIN {X 0,Y 634.664,Z 1229,A -85,B 0,C 180,E1 30528.115,E2 30528.115} C_VEL
LIN {X 0,Y 634.102,Z 1240.475,A -85,B 0,C 180,E1 30526.959,E2 30526.959} C_VEL
LIN {X 0,Y 633.617,Z 1251.131,A -85,B 0,C 180,E1 30525.748,E2 30525.748} C_VEL
LIN {X 0,Y 633.191,Z 1260.279,A -85,B 0,C 180,E1 30524.531,E2 30524.531} C_VEL
LIN {X 0,Y 632.741,Z 1270.509,A -85,B 0,C 180,E1 30522.966,E2 30522.966} C_VEL
LIN {X 0,Y 632.347,Z 1281.586,A -85,B 0,C 180,E1 30520.937,E2 30520.937} C_VEL
LIN {X 0,Y 632.148,Z 1288.982,A -85,B 0,C 180,E1 30519.283,E2 30519.283} C_VEL
LIN {X 0,Y 632.018,Z 1295.058,A -85,B 0,C 180,E1 30517.635,E2 30517.635} C_VEL
LIN {X 0,Y 631.939,Z 1300.898,A -85,B 0,C 180,E1 30515.59,E2 30515.59} C_VEL
LIN {X 0,Y 631.914,Z 1304.518,A -85,B 0,C 180,E1 30513.718,E2 30513.718} C_VEL
LIN {X 0,Y 631.911,Z 1306.588,A -85,B 0,C 180,E1 30511.994,E2 30511.994} C_VEL
LIN {X 0,Y 631.919,Z 1307.5,A -85,B 0,C 180,E1 30509.999,E2 30509.999} C_VEL
LIN {X 0,Y 631.912,Z 1306.585,A -85,B 0,C 180,E1 30508.004,E2 30508.004} C_VEL
LIN {X 0,Y 631.914,Z 1304.512,A -85,B 0,C 180,E1 30506.279,E2 30506.279} C_VEL
LIN {X 0,Y 631.939,Z 1300.893,A -85,B 0,C 180,E1 30504.411,E2 30504.411} C_VEL
LIN {X 0,Y 632.018,Z 1295.053,A -85,B 0,C 180,E1 30502.362,E2 30502.362} C_VEL
LIN {X 0,Y 632.147,Z 1288.972,A -85,B 0,C 180,E1 30500.714,E2 30500.714} C_VEL
LIN {X 0,Y 632.349,Z 1281.571,A -85,B 0,C 180,E1 30499.061,E2 30499.061} C_VEL
LIN {X 0,Y 632.724,Z 1271.075,A -85,B 0,C 180,E1 30497.124,E2 30497.124} C_VEL
LIN {X 0,Y 633.166,Z 1260.855,A -85,B 0,C 180,E1 30495.55,E2 30495.55} C_VEL
LIN {X 0,Y 633.585,Z 1251.87,A -85,B 0,C 180,E1 30494.343,E2 30494.343} C_VEL
LIN {X 0,Y 634.11,Z 1240.551,A -85,B 0,C 180,E1 30493.038,E2 30493.038} C_VEL
LIN {X 0,Y 634.786,Z 1227.197,A -85,B 0,C 180,E1 30491.684,E2 30491.684} C_VEL
LIN {X 0,Y 635.716,Z 1208.89,A -85,B 0,C 180,E1 30490.09,E2 30490.09} C_VEL
LIN {X 0,Y 636.566,Z 1192.566,A -85,B 0,C 180,E1 30488.869,E2 30488.869} C_VEL
LIN {X 0,Y 637.575,Z 1172.612,A -85,B 0,C 180,E1 30487.598,E2 30487.598} C_VEL
LIN {X 0,Y 638.566,Z 1152.481,A -85,B 0,C 180,E1 30486.514,E2 30486.514} C_VEL
LIN {X 0,Y 639.451,Z 1132.302,A -85,B 0,C 180,E1 30485.618,E2 30485.618} C_VEL
LIN {X 0,Y 640.337,Z 1110.585,A -85,B 0,C 180,E1 30484.829,E2 30484.829} C_VEL
LIN {X 0,Y 641.087,Z 1088.933,A -85,B 0,C 180,E1 30484.208,E2 30484.208} C_VEL
LIN {X 0,Y 641.691,Z 1067.065,A -85,B 0,C 180,E1 30483.755,E2 30483.755} C_VEL
LIN {X 0,Y 642.168,Z 1036.801,A -85,B 0,C 180,E1 30483.341,E2 30483.341} C_VEL
LIN {X 0,Y 642.558,Z 1020.583,A -85,B 0,C 180,E1 30483.149,E2 30483.149} C_VEL
LIN {X 0,Y 646.213,Z 1007.627,A -85,B 0,C 180,E1 30482.591,E2 30482.591} C_VEL
LIN {X 0,Y 651.303,Z 992.644,A -85,B 0,C 180,E1 30481.979,E2 30481.979} C_VEL
LIN {X 0,Y 657.473,Z 978.786,A -85,B 0,C 180,E1 30481.475,E2 30481.475} C_VEL
LIN {X 0,Y 663.415,Z 964.898,A -85,B 0,C 180,E1 30480.966,E2 30480.966} C_VEL
LIN {X 0,Y 672.751,Z 947.775,A -85,B 0,C 180,E1 30480.432,E2 30480.432} C_VEL
LIN {X 0,Y 688.388,Z 923.607,A -85,B 0,C 180,E1 30479.797,E2 30479.797} C_VEL
LIN {X 0,Y 715.397,Z 883.963,A -85,B 0,C 180,E1 30478.875,E2 30478.875} C_VEL
LIN {X 0,Y 702.663,Z 879.888,A -85,B 0,C 180,E1 30478.161,E2 30478.161} C_VEL
LIN {X 0,Y 690.919,Z 874.26,A -85,B 0,C 180,E1 30477.38,E2 30477.38} C_VEL
LIN {X 0,Y 680.61,Z 867.282,A -85,B 0,C 180,E1 30476.56,E2 30476.56} C_VEL
LIN {X 0,Y 671.723,Z 859.029,A -85,B 0,C 180,E1 30475.705,E2 30475.705} C_VEL
LIN {X 0,Y 663.829,Z 848.919,A -85,B 0,C 180,E1 30474.767,E2 30474.767} C_VEL
LIN {X 0,Y 657.704,Z 837.82,A -85,B 0,C 180,E1 30473.83,E2 30473.83} C_VEL
LIN {X 0,Y 652.963,Z 825.091,A -85,B 0,C 180,E1 30472.849,E2 30472.849} C_VEL
LIN {X 0,Y 649.613,Z 809.836,A -85,B 0,C 180,E1 30471.773,E2 30471.773} C_VEL
LIN {X 0,Y 647.96,Z 791.351,A -85,B 0,C 180,E1 30470.579,E2 30470.579} C_VEL
LIN {X 0,Y 648.179,Z 768.532,A -85,B 0,C 180,E1 30469.214,E2 30469.214} C_VEL
LIN {X 0,Y 650.716,Z 721.055,A -85,B 0,C 180,E1 30466.435,E2 30466.435} C_VEL
LIN {X 0,Y 652.062,Z 696.774,A -85,B 0,C 180,E1 30464.984,E2 30464.984} C_VEL
LIN {X 0,Y 641.247,Z 672.566,A -85,B 0,C 180,E1 30462.589,E2 30462.589} C_VEL
LIN {X 0,Y 633.773,Z 656.597,A -85,B 0,C 180,E1 30460.9,E2 30460.9} C_VEL
LIN {X 0,Y 632.88,Z 653.834,A -85,B 0,C 180,E1 30460.611,E2 30460.611} C_VEL
LIN {X 0,Y 632.875,Z 653.837,A -85,B 0,C 180,E1 30457.579,E2 30457.579} C_VEL
LIN {X 0,Y 632.908,Z 653.95,A -85,B 0,C 180,E1 30455.393,E2 30455.393} C_VEL
LIN {X 0,Y 638.738,Z 669.96,A -85,B 0,C 180,E1 30453.612,E2 30453.612} C_VEL
LIN {X 0,Y 642.716,Z 684.153,A -85,B 0,C 180,E1 30452.145,E2 30452.145} C_VEL
LIN {X 0,Y 642.211,Z 705.674,A -85,B 0,C 180,E1 30450.395,E2 30450.395} C_VEL
LIN {X 0,Y 646.153,Z 724.076,A -85,B 0,C 180,E1 30449.878,E2 30449.878} C_VEL
LIN {X 0,Y 643.675,Z 851.621,A -85,B 0,C 180,E1 30448.166,E2 30448.166} C_VEL
LIN {X 0,Y 641.851,Z 1007.146,A -85,B 0,C 180,E1 30446.234,E2 30446.234} C_VEL
LIN {X 0,Y 641.331,Z 1029.336,A -85,B 0,C 180,E1 30445.8,E2 30445.8} C_VEL
LIN {X 0,Y 640.678,Z 1051.651,A -85,B 0,C 180,E1 30445.193,E2 30445.193} C_VEL
LIN {X 0,Y 639.906,Z 1072.544,A -85,B 0,C 180,E1 30444.461,E2 30444.461} C_VEL
LIN {X 0,Y 639.044,Z 1091.92,A -85,B 0,C 180,E1 30443.613,E2 30443.613} C_VEL
LIN {X 0,Y 638.064,Z 1111.572,A -85,B 0,C 180,E1 30442.578,E2 30442.578} C_VEL
LIN {X 0,Y 637.116,Z 1129.643,A -85,B 0,C 180,E1 30441.449,E2 30441.449} C_VEL
LIN {X 0,Y 636.139,Z 1146.777,A -85,B 0,C 180,E1 30440.187,E2 30440.187} C_VEL
LIN {X 0,Y 635.21,Z 1162.871,A -85,B 0,C 180,E1 30438.797,E2 30438.797} C_VEL
LIN {X 0,Y 634.341,Z 1178.319,A -85,B 0,C 180,E1 30437.238,E2 30437.238} C_VEL
LIN {X 0,Y 633.627,Z 1191.765,A -85,B 0,C 180,E1 30435.655,E2 30435.655} C_VEL
LIN {X 0,Y 632.983,Z 1205.021,A -85,B 0,C 180,E1 30433.8,E2 30433.8} C_VEL
LIN {X 0,Y 632.544,Z 1215.58,A -85,B 0,C 180,E1 30432.044,E2 30432.044} C_VEL
LIN {X 0,Y 632.261,Z 1224.879,A -85,B 0,C 180,E1 30430.202,E2 30430.202} C_VEL
LIN {X 0,Y 632.065,Z 1232.754,A -85,B 0,C 180,E1 30428.277,E2 30428.277} C_VEL
LIN {X 0,Y 631.968,Z 1238.78,A -85,B 0,C 180,E1 30426.359,E2 30426.359} C_VEL
LIN {X 0,Y 631.922,Z 1243.38,A -85,B 0,C 180,E1 30424.356,E2 30424.356} C_VEL
LIN {X 0,Y 631.905,Z 1246.177,A -85,B 0,C 180,E1 30422.449,E2 30422.449} C_VEL
LIN {X 0,Y 631.913,Z 1247.36,A -85,B 0,C 180,E1 30420.544,E2 30420.544} C_VEL
LIN {X 0,Y 631.905,Z 1247.051,A -85,B 0,C 180,E1 30418.549,E2 30418.549} C_VEL
LIN {X 0,Y 631.904,Z 1245.162,A -85,B 0,C 180,E1 30416.644,E2 30416.644} C_VEL
LIN {X 0,Y 631.937,Z 1241.501,A -85,B 0,C 180,E1 30414.643,E2 30414.643} C_VEL
LIN {X 0,Y 632.005,Z 1236.422,A -85,B 0,C 180,E1 30412.729,E2 30412.729} C_VEL
LIN {X 0,Y 632.126,Z 1229.938,A -85,B 0,C 180,E1 30410.899,E2 30410.899} C_VEL
LIN {X 0,Y 632.359,Z 1221.353,A -85,B 0,C 180,E1 30408.97,E2 30408.97} C_VEL
LIN {X 0,Y 632.715,Z 1211.363,A -85,B 0,C 180,E1 30407.125,E2 30407.125} C_VEL
LIN {X 0,Y 633.215,Z 1199.951,A -85,B 0,C 180,E1 30405.365,E2 30405.365} C_VEL
LIN {X 0,Y 633.859,Z 1187.162,A -85,B 0,C 180,E1 30403.693,E2 30403.693} C_VEL
LIN {X 0,Y 634.628,Z 1173.035,A -85,B 0,C 180,E1 30402.107,E2 30402.107} C_VEL
LIN {X 0,Y 635.548,Z 1157.508,A -85,B 0,C 180,E1 30400.612,E2 30400.612} C_VEL
LIN {X 0,Y 636.559,Z 1140.29,A -85,B 0,C 180,E1 30399.207,E2 30399.207} C_VEL
LIN {X 0,Y 637.586,Z 1122.194,A -85,B 0,C 180,E1 30397.947,E2 30397.947} C_VEL
LIN {X 0,Y 638.662,Z 1102.952,A -85,B 0,C 180,E1 30396.812,E2 30396.812} C_VEL
LIN {X 0,Y 639.674,Z 1082.992,A -85,B 0,C 180,E1 30395.824,E2 30395.824} C_VEL
LIN {X 0,Y 640.577,Z 1063.064,A -85,B 0,C 180,E1 30395.024,E2 30395.024} C_VEL
LIN {X 0,Y 641.398,Z 1041.084,A -85,B 0,C 180,E1 30394.318,E2 30394.318} C_VEL
LIN {X 0,Y 642.077,Z 1019.483,A -85,B 0,C 180,E1 30393.791,E2 30393.791} C_VEL
LIN {X 0,Y 642.547,Z 997.612,A -85,B 0,C 180,E1 30393.42,E2 30393.42} C_VEL
LIN {X 0,Y 644.334,Z 842.302,A -85,B 0,C 180,E1 30391.531,E2 30391.531} C_VEL
LIN {X 0,Y 643.562,Z 834.723,A -85,B 0,C 180,E1 30391.397,E2 30391.397} C_VEL
LIN {X 0,Y 638.318,Z 814.927,A -85,B 0,C 180,E1 30390.891,E2 30390.891} C_VEL
LIN {X 0,Y 637.723,Z 808.417,A -85,B 0,C 180,E1 30390.776,E2 30390.776} C_VEL
LIN {X 0,Y 638.926,Z 724.239,A -85,B 0,C 180,E1 30389.686,E2 30389.686} C_VEL
LIN {X 0,Y 633.873,Z 701.983,A -85,B 0,C 180,E1 30389.107,E2 30389.107} C_VEL
LIN {X 0,Y 634.449,Z 684.996,A -85,B 0,C 180,E1 30387.644,E2 30387.644} C_VEL
LIN {X 0,Y 628.2,Z 664.84,A -85,B 0,C 180,E1 30385.484,E2 30385.484} C_VEL
LIN {X 0,Y 624.942,Z 654.826,A -85,B 0,C 180,E1 30384.37,E2 30384.37} C_VEL
LIN {X 0,Y 624.945,Z 654.823,A -85,B 0,C 180,E1 30381.157,E2 30381.157} C_VEL
LIN {X 0,Y 624.954,Z 654.821,A -85,B 0,C 180,E1 30377.904,E2 30377.904} C_VEL
LIN {X 0,Y 624.947,Z 654.823,A -85,B 0,C 180,E1 30374.603,E2 30374.603} C_VEL
LIN {X 0,Y 624.943,Z 654.829,A -85,B 0,C 180,E1 30371.376,E2 30371.376} C_VEL
LIN {X 0,Y 624.943,Z 654.825,A -85,B 0,C 180,E1 30368.225,E2 30368.225} C_VEL
LIN {X 0,Y 624.939,Z 654.821,A -85,B 0,C 180,E1 30365.058,E2 30365.058} C_VEL
LIN {X 0,Y 624.94,Z 654.82,A -85,B 0,C 180,E1 30361.979,E2 30361.979} C_VEL
LIN {X 0,Y 624.948,Z 654.825,A -85,B 0,C 180,E1 30358.895,E2 30358.895} C_VEL
LIN {X 0,Y 624.943,Z 654.822,A -85,B 0,C 180,E1 30355.738,E2 30355.738} C_VEL
LIN {X 0,Y 624.94,Z 654.82,A -85,B 0,C 180,E1 30352.582,E2 30352.582} C_VEL
LIN {X 0,Y 624.938,Z 654.819,A -85,B 0,C 180,E1 30349.44,E2 30349.44} C_VEL
LIN {X 0,Y 624.94,Z 654.826,A -85,B 0,C 180,E1 30346.356,E2 30346.356} C_VEL
LIN {X 0,Y 624.942,Z 654.82,A -85,B 0,C 180,E1 30343.227,E2 30343.227} C_VEL
LIN {X 0,Y 624.938,Z 654.82,A -85,B 0,C 180,E1 30340.045,E2 30340.045} C_VEL
LIN {X 0,Y 624.935,Z 654.82,A -85,B 0,C 180,E1 30336.893,E2 30336.893} C_VEL
LIN {X 0,Y 624.936,Z 654.822,A -85,B 0,C 180,E1 30333.762,E2 30333.762} C_VEL
LIN {X 0,Y 624.941,Z 654.825,A -85,B 0,C 180,E1 30330.643,E2 30330.643} C_VEL
LIN {X 0,Y 624.937,Z 654.821,A -85,B 0,C 180,E1 30327.525,E2 30327.525} C_VEL
LIN {X 0,Y 624.936,Z 654.82,A -85,B 0,C 180,E1 30324.383,E2 30324.383} C_VEL
LIN {X 0,Y 624.938,Z 654.825,A -85,B 0,C 180,E1 30321.351,E2 30321.351} C_VEL
LIN {X 0,Y 624.944,Z 654.82,A -85,B 0,C 180,E1 30318.184,E2 30318.184} C_VEL
LIN {X 0,Y 624.939,Z 654.818,A -85,B 0,C 180,E1 30315.074,E2 30315.074} C_VEL
LIN {X 0,Y 624.935,Z 654.821,A -85,B 0,C 180,E1 30311.918,E2 30311.918} C_VEL
LIN {X 0,Y 624.937,Z 654.825,A -85,B 0,C 180,E1 30308.803,E2 30308.803} C_VEL
LIN {X 0,Y 624.945,Z 654.825,A -85,B 0,C 180,E1 30305.722,E2 30305.722} C_VEL
LIN {X 0,Y 624.939,Z 654.819,A -85,B 0,C 180,E1 30302.564,E2 30302.564} C_VEL
LIN {X 0,Y 624.939,Z 654.822,A -85,B 0,C 180,E1 30299.525,E2 30299.525} C_VEL
LIN {X 0,Y 624.939,Z 654.827,A -85,B 0,C 180,E1 30296.388,E2 30296.388} C_VEL
LIN {X 0,Y 624.944,Z 654.82,A -85,B 0,C 180,E1 30293.248,E2 30293.248} C_VEL
LIN {X 0,Y 624.94,Z 654.822,A -85,B 0,C 180,E1 30290.092,E2 30290.092} C_VEL
LIN {X 0,Y 624.938,Z 654.825,A -85,B 0,C 180,E1 30286.987,E2 30286.987} C_VEL
LIN {X 0,Y 624.956,Z 654.921,A -85,B 0,C 180,E1 30284.42,E2 30284.42} C_VEL
LIN {X 0,Y 634.442,Z 681.598,A -85,B 0,C 180,E1 30281.669,E2 30281.669} C_VEL
LIN {X 0,Y 636.888,Z 689.532,A -85,B 0,C 180,E1 30280.895,E2 30280.895} C_VEL
LIN {X 0,Y 635.183,Z 728.254,A -85,B 0,C 180,E1 30277.989,E2 30277.989} C_VEL
LIN {X 0,Y 633.257,Z 771.396,A -85,B 0,C 180,E1 30274.812,E2 30274.812} C_VEL
LIN {X 0,Y 631.456,Z 815.862,A -85,B 0,C 180,E1 30271.584,E2 30271.584} C_VEL
LIN {X 0,Y 629.707,Z 863.902,A -85,B 0,C 180,E1 30268.138,E2 30268.138} C_VEL
LIN {X 0,Y 628.709,Z 898.39,A -85,B 0,C 180,E1 30265.721,E2 30265.721} C_VEL
LIN {X 0,Y 629.415,Z 906.069,A -85,B 0,C 180,E1 30265.59,E2 30265.59} C_VEL
LIN {X 0,Y 627.659,Z 1042.148,A -85,B 0,C 180,E1 30263.731,E2 30263.731} C_VEL
LIN {X 0,Y 627.431,Z 1059.245,A -85,B 0,C 180,E1 30263.314,E2 30263.314} C_VEL
LIN {X 0,Y 627.105,Z 1074.553,A -85,B 0,C 180,E1 30262.766,E2 30262.766} C_VEL
LIN {X 0,Y 626.678,Z 1090.054,A -85,B 0,C 180,E1 30262.021,E2 30262.021} C_VEL
LIN {X 0,Y 626.263,Z 1103.481,A -85,B 0,C 180,E1 30261.192,E2 30261.192} C_VEL
LIN {X 0,Y 625.805,Z 1117.001,A -85,B 0,C 180,E1 30260.14,E2 30260.14} C_VEL
LIN {X 0,Y 625.413,Z 1128.367,A -85,B 0,C 180,E1 30259.035,E2 30259.035} C_VEL
LIN {X 0,Y 625.047,Z 1138.627,A -85,B 0,C 180,E1 30257.791,E2 30257.791} C_VEL
LIN {X 0,Y 624.785,Z 1146.823,A -85,B 0,C 180,E1 30256.547,E2 30256.547} C_VEL
LIN {X 0,Y 624.571,Z 1154.007,A -85,B 0,C 180,E1 30255.127,E2 30255.127} C_VEL
LIN {X 0,Y 624.457,Z 1159.311,A -85,B 0,C 180,E1 30253.708,E2 30253.708} C_VEL
LIN {X 0,Y 624.394,Z 1162.989,A -85,B 0,C 180,E1 30252.203,E2 30252.203} C_VEL
LIN {X 0,Y 624.372,Z 1164.903,A -85,B 0,C 180,E1 30250.706,E2 30250.706} C_VEL
LIN {X 0,Y 624.388,Z 1165.055,A -85,B 0,C 180,E1 30249.215,E2 30249.215} C_VEL
LIN {X 0,Y 624.455,Z 1163.344,A -85,B 0,C 180,E1 30247.637,E2 30247.637} C_VEL
LIN {X 0,Y 624.553,Z 1159.937,A -85,B 0,C 180,E1 30246.158,E2 30246.158} C_VEL
LIN {X 0,Y 624.726,Z 1154.677,A -85,B 0,C 180,E1 30244.682,E2 30244.682} C_VEL
LIN {X 0,Y 624.987,Z 1147.894,A -85,B 0,C 180,E1 30243.302,E2 30243.302} C_VEL
LIN {X 0,Y 625.352,Z 1139.02,A -85,B 0,C 180,E1 30241.924,E2 30241.924} C_VEL
LIN {X 0,Y 625.771,Z 1129.31,A -85,B 0,C 180,E1 30240.732,E2 30240.732} C_VEL
LIN {X 0,Y 626.271,Z 1117.135,A -85,B 0,C 180,E1 30239.543,E2 30239.543} C_VEL
LIN {X 0,Y 626.752,Z 1104.87,A -85,B 0,C 180,E1 30238.583,E2 30238.583} C_VEL
LIN {X 0,Y 627.222,Z 1090.945,A -85,B 0,C 180,E1 30237.716,E2 30237.716} C_VEL
LIN {X 0,Y 627.665,Z 1076.959,A -85,B 0,C 180,E1 30237.032,E2 30237.032} C_VEL
LIN {X 0,Y 627.991,Z 1061.29,A -85,B 0,C 180,E1 30236.463,E2 30236.463} C_VEL
LIN {X 0,Y 628.209,Z 1045.137,A -85,B 0,C 180,E1 30236.053,E2 30236.053} C_VEL
LIN {X 0,Y 631.331,Z 904.878,A -85,B 0,C 180,E1 30233.817,E2 30233.817} C_VEL
LIN {X 0,Y 633.873,Z 860.388,A -85,B 0,C 180,E1 30230.466,E2 30230.466} C_VEL
LIN {X 0,Y 636.934,Z 816.496,A -85,B 0,C 180,E1 30227.073,E2 30227.073} C_VEL
LIN {X 0,Y 640.686,Z 773.866,A -85,B 0,C 180,E1 30223.685,E2 30223.685} C_VEL
LIN {X 0,Y 645.09,Z 733.356,A -85,B 0,C 180,E1 30220.345,E2 30220.345} C_VEL
LIN {X 0,Y 648.004,Z 705.728,A -85,B 0,C 180,E1 30217.907,E2 30217.907} C_VEL
LIN {X 0,Y 643.339,Z 693.092,A -85,B 0,C 180,E1 30215.97,E2 30215.97} C_VEL
LIN {X 0,Y 638.868,Z 682.348,A -85,B 0,C 180,E1 30214.009,E2 30214.009} C_VEL
LIN {X 0,Y 636.461,Z 677.309,A -85,B 0,C 180,E1 30212.897,E2 30212.897} C_VEL
LIN {X 0,Y 634.875,Z 673.855,A -85,B 0,C 180,E1 30212.068,E2 30212.068} C_VEL
LIN {X 0,Y 633.06,Z 669.893,A -85,B 0,C 180,E1 30210.994,E2 30210.994} C_VEL
LIN {X 0,Y 631.112,Z 666.087,A -85,B 0,C 180,E1 30209.703,E2 30209.703} C_VEL
LIN {X 0,Y 630.392,Z 664.899,A -85,B 0,C 180,E1 30209.181,E2 30209.181} C_VEL
LIN {X 0,Y 628.542,Z 661.692,A -85,B 0,C 180,E1 30207.257,E2 30207.257} C_VEL
LIN {X 0,Y 628.228,Z 660.346,A -85,B 0,C 180,E1 30205.927,E2 30205.927} C_VEL
LIN {X 0,Y 628.427,Z 660.735,A -85,B 0,C 180,E1 30204.235,E2 30204.235} C_VEL
LIN {X 0,Y 629.502,Z 663.684,A -85,B 0,C 180,E1 30202.415,E2 30202.415} C_VEL
LIN {X 0,Y 631.399,Z 665.91,A -85,B 0,C 180,E1 30201.279,E2 30201.279} C_VEL
LIN {X 0,Y 632.838,Z 669.369,A -85,B 0,C 180,E1 30200.303,E2 30200.303} C_VEL
LIN {X 0,Y 634.079,Z 671.312,A -85,B 0,C 180,E1 30199.747,E2 30199.747} C_VEL
LIN {X 0,Y 636.614,Z 676.479,A -85,B 0,C 180,E1 30198.605,E2 30198.605} C_VEL
LIN {X 0,Y 639.88,Z 683.092,A -85,B 0,C 180,E1 30197.388,E2 30197.388} C_VEL
LIN {X 0,Y 644.367,Z 693.775,A -85,B 0,C 180,E1 30195.834,E2 30195.834} C_VEL
LIN {X 0,Y 646.339,Z 699.155,A -85,B 0,C 180,E1 30195.169,E2 30195.169} C_VEL
LIN {X 0,Y 641.525,Z 739.522,A -85,B 0,C 180,E1 30192.563,E2 30192.563} C_VEL
LIN {X 0,Y 638.494,Z 779.081,A -85,B 0,C 180,E1 30190.125,E2 30190.125} C_VEL
LIN {X 0,Y 638.958,Z 799.566,A -85,B 0,C 180,E1 30188.802,E2 30188.802} C_VEL
LIN {X 0,Y 641.002,Z 815.158,A -85,B 0,C 180,E1 30187.733,E2 30187.733} C_VEL
LIN {X 0,Y 644.926,Z 830.042,A -85,B 0,C 180,E1 30186.646,E2 30186.646} C_VEL
LIN {X 0,Y 650.625,Z 843.283,A -85,B 0,C 180,E1 30185.612,E2 30185.612} C_VEL
LIN {X 0,Y 657.74,Z 854.628,A -85,B 0,C 180,E1 30184.671,E2 30184.671} C_VEL
LIN {X 0,Y 665.734,Z 864.039,A -85,B 0,C 180,E1 30183.842,E2 30183.842} C_VEL
LIN {X 0,Y 675.932,Z 873.081,A -85,B 0,C 180,E1 30182.991,E2 30182.991} C_VEL
LIN {X 0,Y 687.693,Z 880.812,A -85,B 0,C 180,E1 30182.197,E2 30182.197} C_VEL
LIN {X 0,Y 700.988,Z 887.108,A -85,B 0,C 180,E1 30181.461,E2 30181.461} C_VEL
LIN {X 0,Y 704.282,Z 888.456,A -85,B 0,C 180,E1 30181.294,E2 30181.294} C_VEL
LIN {X 0,Y 670.672,Z 936.51,A -85,B 0,C 180,E1 30180.016,E2 30180.016} C_VEL
LIN {X 0,Y 659.346,Z 955.296,A -85,B 0,C 180,E1 30179.427,E2 30179.427} C_VEL
LIN {X 0,Y 651.96,Z 970.509,A -85,B 0,C 180,E1 30178.887,E2 30178.887} C_VEL
LIN {X 0,Y 648.099,Z 980.036,A -85,B 0,C 180,E1 30178.52,E2 30178.52} C_VEL
LIN {X 0,Y 642.051,Z 993.719,A -85,B 0,C 180,E1 30178.002,E2 30178.002} C_VEL
LIN {X 0,Y 635.281,Z 1015.549,A -85,B 0,C 180,E1 30177.091,E2 30177.091} C_VEL
LIN {X 0,Y 634.532,Z 1030.124,A -85,B 0,C 180,E1 30176.937,E2 30176.937} C_VEL
LIN {X 0,Y 634.037,Z 1065.459,A -85,B 0,C 180,E1 30176.469,E2 30176.469} C_VEL
LIN {X 0,Y 633.4,Z 1087.709,A -85,B 0,C 180,E1 30176.01,E2 30176.01} C_VEL
LIN {X 0,Y 632.641,Z 1109.13,A -85,B 0,C 180,E1 30175.398,E2 30175.398} C_VEL
LIN {X 0,Y 631.693,Z 1130.967,A -85,B 0,C 180,E1 30174.599,E2 30174.599} C_VEL
LIN {X 0,Y 630.722,Z 1152.004,A -85,B 0,C 180,E1 30173.644,E2 30173.644} C_VEL
LIN {X 0,Y 629.624,Z 1172.763,A -85,B 0,C 180,E1 30172.501,E2 30172.501} C_VEL
LIN {X 0,Y 628.584,Z 1192.075,A -85,B 0,C 180,E1 30171.227,E2 30171.227} C_VEL
LIN {X 0,Y 627.608,Z 1211.218,A -85,B 0,C 180,E1 30169.787,E2 30169.787} C_VEL
LIN {X 0,Y 626.818,Z 1226.69,A -85,B 0,C 180,E1 30168.41,E2 30168.41} C_VEL
LIN {X 0,Y 626.203,Z 1238.898,A -85,B 0,C 180,E1 30167.18,E2 30167.18} C_VEL
LIN {X 0,Y 625.689,Z 1249.707,A -85,B 0,C 180,E1 30165.952,E2 30165.952} C_VEL
LIN {X 0,Y 625.223,Z 1259.977,A -85,B 0,C 180,E1 30164.635,E2 30164.635} C_VEL
LIN {X 0,Y 624.8,Z 1270.216,A -85,B 0,C 180,E1 30163.134,E2 30163.134} C_VEL
LIN {X 0,Y 624.437,Z 1280.268,A -85,B 0,C 180,E1 30161.358,E2 30161.358} C_VEL
LIN {X 0,Y 624.192,Z 1288.23,A -85,B 0,C 180,E1 30159.589,E2 30159.589} C_VEL
LIN {X 0,Y 624.046,Z 1294.119,A -85,B 0,C 180,E1 30158.012,E2 30158.012} C_VEL
LIN {X 0,Y 623.966,Z 1299.129,A -85,B 0,C 180,E1 30156.347,E2 30156.347} C_VEL
LIN {X 0,Y 623.923,Z 1303.681,A -85,B 0,C 180,E1 30154.318,E2 30154.318} C_VEL
LIN {X 0,Y 623.907,Z 1306.253,A -85,B 0,C 180,E1 30152.387,E2 30152.387} C_VEL
LIN {X 0,Y 623.909,Z 1307.295,A -85,B 0,C 180,E1 30150.733,E2 30150.733} C_VEL
LIN {X 0,Y 623.916,Z 1307.238,A -85,B 0,C 180,E1 30149.081,E2 30149.081} C_VEL
LIN {X 0,Y 623.918,Z 1305.731,A -85,B 0,C 180,E1 30147.059,E2 30147.059} C_VEL
LIN {X 0,Y 623.924,Z 1302.556,A -85,B 0,C 180,E1 30145.126,E2 30145.126} C_VEL
LIN {X 0,Y 623.968,Z 1298.618,A -85,B 0,C 180,E1 30143.466,E2 30143.466} C_VEL
LIN {X 0,Y 624.059,Z 1293.798,A -85,B 0,C 180,E1 30141.893,E2 30141.893} C_VEL
LIN {X 0,Y 624.239,Z 1286.72,A -85,B 0,C 180,E1 30140.037,E2 30140.037} C_VEL
LIN {X 0,Y 624.53,Z 1277.8,A -85,B 0,C 180,E1 30138.173,E2 30138.173} C_VEL
LIN {X 0,Y 624.852,Z 1269.01,A -85,B 0,C 180,E1 30136.677,E2 30136.677} C_VEL
LIN {X 0,Y 625.289,Z 1258.724,A -85,B 0,C 180,E1 30135.175,E2 30135.175} C_VEL
LIN {X 0,Y 625.894,Z 1246.103,A -85,B 0,C 180,E1 30133.574,E2 30133.574} C_VEL
LIN {X 0,Y 626.639,Z 1231.208,A -85,B 0,C 180,E1 30131.967,E2 30131.967} C_VEL
LIN {X 0,Y 627.38,Z 1217.152,A -85,B 0,C 180,E1 30130.649,E2 30130.649} C_VEL
LIN {X 0,Y 628.253,Z 1201.495,A -85,B 0,C 180,E1 30129.363,E2 30129.363} C_VEL
LIN {X 0,Y 629.229,Z 1183.208,A -85,B 0,C 180,E1 30128.072,E2 30128.072} C_VEL
LIN {X 0,Y 630.268,Z 1164.313,A -85,B 0,C 180,E1 30126.929,E2 30126.929} C_VEL
LIN {X 0,Y 631.218,Z 1144.495,A -85,B 0,C 180,E1 30125.929,E2 30125.929} C_VEL
LIN {X 0,Y 632.236,Z 1122.806,A -85,B 0,C 180,E1 30125.022,E2 30125.022} C_VEL
LIN {X 0,Y 633.117,Z 1101.655,A -85,B 0,C 180,E1 30124.308,E2 30124.308} C_VEL
LIN {X 0,Y 633.846,Z 1080.148,A -85,B 0,C 180,E1 30123.757,E2 30123.757} C_VEL
LIN {X 0,Y 634.455,Z 1057.268,A -85,B 0,C 180,E1 30123.335,E2 30123.335} C_VEL
LIN {X 0,Y 635.235,Z 1019.826,A -85,B 0,C 180,E1 30122.865,E2 30122.865} C_VEL
LIN {X 0,Y 638.928,Z 1006.89,A -85,B 0,C 180,E1 30122.303,E2 30122.303} C_VEL
LIN {X 0,Y 643.952,Z 992.164,A -85,B 0,C 180,E1 30121.692,E2 30121.692} C_VEL
LIN {X 0,Y 650.564,Z 977.25,A -85,B 0,C 180,E1 30121.144,E2 30121.144} C_VEL
LIN {X 0,Y 656.981,Z 962.503,A -85,B 0,C 180,E1 30120.604,E2 30120.604} C_VEL
LIN {X 0,Y 666.872,Z 944.615,A -85,B 0,C 180,E1 30120.046,E2 30120.046} C_VEL
LIN {X 0,Y 683.364,Z 919.313,A -85,B 0,C 180,E1 30119.389,E2 30119.389} C_VEL
LIN {X 0,Y 704.338,Z 888.552,A -85,B 0,C 180,E1 30118.663,E2 30118.663} C_VEL
LIN {X 0,Y 691.749,Z 883.478,A -85,B 0,C 180,E1 30117.891,E2 30117.891} C_VEL
LIN {X 0,Y 680.337,Z 876.88,A -85,B 0,C 180,E1 30117.056,E2 30117.056} C_VEL
LIN {X 0,Y 670.365,Z 868.966,A -85,B 0,C 180,E1 30116.181,E2 30116.181} C_VEL
LIN {X 0,Y 661.837,Z 859.788,A -85,B 0,C 180,E1 30115.272,E2 30115.272} C_VEL
LIN {X 0,Y 654.212,Z 848.388,A -85,B 0,C 180,E1 30114.251,E2 30114.251} C_VEL
LIN {X 0,Y 648.6,Z 836.252,A -85,B 0,C 180,E1 30113.262,E2 30113.262} C_VEL
LIN {X 0,Y 644.447,Z 822.425,A -85,B 0,C 180,E1 30112.227,E2 30112.227} C_VEL
LIN {X 0,Y 641.872,Z 806.951,A -85,B 0,C 180,E1 30111.159,E2 30111.159} C_VEL
LIN {X 0,Y 640.816,Z 786.651,A -85,B 0,C 180,E1 30109.869,E2 30109.869} C_VEL
LIN {X 0,Y 644.233,Z 718.256,A -85,B 0,C 180,E1 30105.812,E2 30105.812} C_VEL
LIN {X 0,Y 645.236,Z 700.146,A -85,B 0,C 180,E1 30104.712,E2 30104.712} C_VEL
LIN {X 0,Y 633.687,Z 674.269,A -85,B 0,C 180,E1 30102.114,E2 30102.114} C_VEL
LIN {X 0,Y 626.173,Z 658.201,A -85,B 0,C 180,E1 30100.386,E2 30100.386} C_VEL
LIN {X 0,Y 624.954,Z 654.824,A -85,B 0,C 180,E1 30100.029,E2 30100.029} C_VEL
LIN {X 0,Y 624.953,Z 654.825,A -85,B 0,C 180,E1 30096.869,E2 30096.869} C_VEL
LIN {X 0,Y 624.977,Z 655.035,A -85,B 0,C 180,E1 30095.981,E2 30095.981} C_VEL
LIN {X 0,Y 630.91,Z 670.369,A -85,B 0,C 180,E1 30094.178,E2 30094.178} C_VEL
LIN {X 0,Y 635.78,Z 686.945,A -85,B 0,C 180,E1 30092.405,E2 30092.405} C_VEL
LIN {X 0,Y 635.264,Z 706.378,A -85,B 0,C 180,E1 30090.806,E2 30090.806} C_VEL
LIN {X 0,Y 639.346,Z 725.48,A -85,B 0,C 180,E1 30090.241,E2 30090.241} C_VEL
LIN {X 0,Y 636.595,Z 847.445,A -85,B 0,C 180,E1 30088.544,E2 30088.544} C_VEL
LIN {X 0,Y 634.788,Z 979.552,A -85,B 0,C 180,E1 30086.864,E2 30086.864} C_VEL
LIN {X 0,Y 634.353,Z 1010.893,A -85,B 0,C 180,E1 30086.445,E2 30086.445} C_VEL
LIN {X 0,Y 633.801,Z 1033.208,A -85,B 0,C 180,E1 30085.975,E2 30085.975} C_VEL
LIN {X 0,Y 633.092,Z 1054.36,A -85,B 0,C 180,E1 30085.37,E2 30085.37} C_VEL
LIN {X 0,Y 632.28,Z 1074.929,A -85,B 0,C 180,E1 30084.622,E2 30084.622} C_VEL
LIN {X 0,Y 631.353,Z 1095.024,A -85,B 0,C 180,E1 30083.72,E2 30083.72} C_VEL
LIN {X 0,Y 630.33,Z 1114.209,A -85,B 0,C 180,E1 30082.673,E2 30082.673} C_VEL
LIN {X 0,Y 629.247,Z 1133.28,A -85,B 0,C 180,E1 30081.437,E2 30081.437} C_VEL
LIN {X 0,Y 628.263,Z 1150.097,A -85,B 0,C 180,E1 30080.155,E2 30080.155} C_VEL
LIN {X 0,Y 627.31,Z 1165.58,A -85,B 0,C 180,E1 30078.773,E2 30078.773} C_VEL
LIN {X 0,Y 626.454,Z 1180.02,A -85,B 0,C 180,E1 30077.27,E2 30077.27} C_VEL
LIN {X 0,Y 625.71,Z 1193.277,A -85,B 0,C 180,E1 30075.668,E2 30075.668} C_VEL
LIN {X 0,Y 625.093,Z 1205.142,A -85,B 0,C 180,E1 30073.977,E2 30073.977} C_VEL
LIN {X 0,Y 624.611,Z 1215.638,A -85,B 0,C 180,E1 30072.199,E2 30072.199} C_VEL
LIN {X 0,Y 624.281,Z 1225.283,A -85,B 0,C 180,E1 30070.241,E2 30070.241} C_VEL
LIN {X 0,Y 624.075,Z 1233.103,A -85,B 0,C 180,E1 30068.291,E2 30068.291} C_VEL
LIN {X 0,Y 623.97,Z 1239.034,A -85,B 0,C 180,E1 30066.348,E2 30066.348} C_VEL
LIN {X 0,Y 623.921,Z 1243.539,A -85,B 0,C 180,E1 30064.32,E2 30064.32} C_VEL
LIN {X 0,Y 623.903,Z 1246.289,A -85,B 0,C 180,E1 30062.388,E2 30062.388} C_VEL
LIN {X 0,Y 623.91,Z 1247.383,A -85,B 0,C 180,E1 30060.459,E2 30060.459} C_VEL
LIN {X 0,Y 623.909,Z 1246.982,A -85,B 0,C 180,E1 30058.439,E2 30058.439} C_VEL
LIN {X 0,Y 623.909,Z 1245.048,A -85,B 0,C 180,E1 30056.509,E2 30056.509} C_VEL
LIN {X 0,Y 623.941,Z 1241.499,A -85,B 0,C 180,E1 30054.575,E2 30054.575} C_VEL
LIN {X 0,Y 624.013,Z 1236.419,A -85,B 0,C 180,E1 30052.635,E2 30052.635} C_VEL
LIN {X 0,Y 624.147,Z 1229.936,A -85,B 0,C 180,E1 30050.781,E2 30050.781} C_VEL
LIN {X 0,Y 624.402,Z 1221.349,A -85,B 0,C 180,E1 30048.827,E2 30048.827} C_VEL
LIN {X 0,Y 624.794,Z 1211.424,A -85,B 0,C 180,E1 30046.959,E2 30046.959} C_VEL
LIN {X 0,Y 625.347,Z 1200.059,A -85,B 0,C 180,E1 30045.177,E2 30045.177} C_VEL
LIN {X 0,Y 626.042,Z 1187.21,A -85,B 0,C 180,E1 30043.483,E2 30043.483} C_VEL
LIN {X 0,Y 626.928,Z 1172.082,A -85,B 0,C 180,E1 30041.784,E2 30041.784} C_VEL
LIN {X 0,Y 627.873,Z 1156.843,A -85,B 0,C 180,E1 30040.317,E2 30040.317} C_VEL
LIN {X 0,Y 628.928,Z 1140.113,A -85,B 0,C 180,E1 30038.943,E2 30038.943} C_VEL
LIN {X 0,Y 629.989,Z 1122.504,A -85,B 0,C 180,E1 30037.708,E2 30037.708} C_VEL
LIN {X 0,Y 631.118,Z 1103.409,A -85,B 0,C 180,E1 30036.568,E2 30036.568} C_VEL
LIN {X 0,Y 632.193,Z 1083.481,A -85,B 0,C 180,E1 30035.569,E2 30035.569} C_VEL
LIN {X 0,Y 633.146,Z 1063.608,A -85,B 0,C 180,E1 30034.761,E2 30034.761} C_VEL
LIN {X 0,Y 634.026,Z 1041.514,A -85,B 0,C 180,E1 30034.04,E2 30034.04} C_VEL
LIN {X 0,Y 634.749,Z 1019.824,A -85,B 0,C 180,E1 30033.504,E2 30033.504} C_VEL
LIN {X 0,Y 635.254,Z 997.773,A -85,B 0,C 180,E1 30033.126,E2 30033.126} C_VEL
LIN {X 0,Y 637.723,Z 808.417,A -85,B 0,C 180,E1 30030.776,E2 30030.776} C_VEL
LIN {X 0,Y 636.952,Z 800.848,A -85,B 0,C 180,E1 30030.635,E2 30030.635} C_VEL
LIN {X 0,Y 631.823,Z 781.078,A -85,B 0,C 180,E1 30030.107,E2 30030.107} C_VEL
LIN {X 0,Y 631.283,Z 774.571,A -85,B 0,C 180,E1 30029.989,E2 30029.989} C_VEL
LIN {X 0,Y 631.98,Z 725.69,A -85,B 0,C 180,E1 30029.34,E2 30029.34} C_VEL
LIN {X 0,Y 626.654,Z 702.144,A -85,B 0,C 180,E1 30028.71,E2 30028.71} C_VEL
LIN {X 0,Y 627.22,Z 688.051,A -85,B 0,C 180,E1 30027.492,E2 30027.492} C_VEL
LIN {X 0,Y 620.575,Z 666.635,A -85,B 0,C 180,E1 30025.178,E2 30025.178} C_VEL
LIN {X 0,Y 617.013,Z 655.811,A -85,B 0,C 180,E1 30023.965,E2 30023.965} C_VEL
LIN {X 0,Y 617.005,Z 655.812,A -85,B 0,C 180,E1 30020.772,E2 30020.772} C_VEL
LIN {X 0,Y 617.003,Z 655.811,A -85,B 0,C 180,E1 30017.611,E2 30017.611} C_VEL
LIN {X 0,Y 617.001,Z 655.812,A -85,B 0,C 180,E1 30014.435,E2 30014.435} C_VEL
LIN {X 0,Y 616.998,Z 655.816,A -85,B 0,C 180,E1 30011.24,E2 30011.24} C_VEL
LIN {X 0,Y 617.003,Z 655.815,A -85,B 0,C 180,E1 30008.13,E2 30008.13} C_VEL
LIN {X 0,Y 616.999,Z 655.81,A -85,B 0,C 180,E1 30005.008,E2 30005.008} C_VEL
LIN {X 0,Y 616.997,Z 655.809,A -85,B 0,C 180,E1 30001.877,E2 30001.877} C_VEL
LIN {X 0,Y 617,Z 655.813,A -85,B 0,C 180,E1 29998.749,E2 29998.749} C_VEL
LIN {X 0,Y 617.004,Z 655.812,A -85,B 0,C 180,E1 29995.639,E2 29995.639} C_VEL
LIN {X 0,Y 616.997,Z 655.81,A -85,B 0,C 180,E1 29992.487,E2 29992.487} C_VEL
LIN {X 0,Y 616.998,Z 655.807,A -85,B 0,C 180,E1 29989.404,E2 29989.404} C_VEL
LIN {X 0,Y 616.998,Z 655.814,A -85,B 0,C 180,E1 29986.283,E2 29986.283} C_VEL
LIN {X 0,Y 617.003,Z 655.809,A -85,B 0,C 180,E1 29983.21,E2 29983.21} C_VEL
LIN {X 0,Y 617,Z 655.808,A -85,B 0,C 180,E1 29980.081,E2 29980.081} C_VEL
LIN {X 0,Y 617.001,Z 655.809,A -85,B 0,C 180,E1 29976.982,E2 29976.982} C_VEL
LIN {X 0,Y 616.999,Z 655.81,A -85,B 0,C 180,E1 29973.811,E2 29973.811} C_VEL
LIN {X 0,Y 617.002,Z 655.814,A -85,B 0,C 180,E1 29970.651,E2 29970.651} C_VEL
LIN {X 0,Y 616.998,Z 655.81,A -85,B 0,C 180,E1 29967.494,E2 29967.494} C_VEL
LIN {X 0,Y 616.996,Z 655.809,A -85,B 0,C 180,E1 29964.328,E2 29964.328} C_VEL
LIN {X 0,Y 616.996,Z 655.813,A -85,B 0,C 180,E1 29961.239,E2 29961.239} C_VEL
LIN {X 0,Y 617.007,Z 655.81,A -85,B 0,C 180,E1 29958.125,E2 29958.125} C_VEL
LIN {X 0,Y 616.998,Z 655.808,A -85,B 0,C 180,E1 29954.974,E2 29954.974} C_VEL
LIN {X 0,Y 616.996,Z 655.81,A -85,B 0,C 180,E1 29951.873,E2 29951.873} C_VEL
LIN {X 0,Y 616.998,Z 655.813,A -85,B 0,C 180,E1 29948.717,E2 29948.717} C_VEL
LIN {X 0,Y 617.01,Z 655.814,A -85,B 0,C 180,E1 29945.593,E2 29945.593} C_VEL
LIN {X 0,Y 617.002,Z 655.81,A -85,B 0,C 180,E1 29942.39,E2 29942.39} C_VEL
LIN {X 0,Y 616.998,Z 655.811,A -85,B 0,C 180,E1 29939.306,E2 29939.306} C_VEL
LIN {X 0,Y 616.998,Z 655.816,A -85,B 0,C 180,E1 29936.232,E2 29936.232} C_VEL
LIN {X 0,Y 617.008,Z 655.81,A -85,B 0,C 180,E1 29933.161,E2 29933.161} C_VEL
LIN {X 0,Y 617.001,Z 655.811,A -85,B 0,C 180,E1 29930.043,E2 29930.043} C_VEL
LIN {X 0,Y 616.999,Z 655.814,A -85,B 0,C 180,E1 29926.96,E2 29926.96} C_VEL
LIN {X 0,Y 617.001,Z 655.831,A -85,B 0,C 180,E1 29924.884,E2 29924.884} C_VEL
LIN {X 0,Y 626.868,Z 683.463,A -85,B 0,C 180,E1 29921.99,E2 29921.99} C_VEL
LIN {X 0,Y 629.718,Z 692.45,A -85,B 0,C 180,E1 29921.1,E2 29921.1} C_VEL
LIN {X 0,Y 627.921,Z 730.511,A -85,B 0,C 180,E1 29918.217,E2 29918.217} C_VEL
LIN {X 0,Y 625.892,Z 773.077,A -85,B 0,C 180,E1 29915.052,E2 29915.052} C_VEL
LIN {X 0,Y 623.972,Z 818.026,A -85,B 0,C 180,E1 29911.763,E2 29911.763} C_VEL
LIN {X 0,Y 622.147,Z 865.944,A -85,B 0,C 180,E1 29908.302,E2 29908.302} C_VEL
LIN {X 0,Y 621.125,Z 899.09,A -85,B 0,C 180,E1 29905.958,E2 29905.958} C_VEL
LIN {X 0,Y 621.852,Z 906.852,A -85,B 0,C 180,E1 29905.823,E2 29905.823} C_VEL
LIN {X 0,Y 619.947,Z 1043.033,A -85,B 0,C 180,E1 29903.915,E2 29903.915} C_VEL
LIN {X 0,Y 619.703,Z 1060.221,A -85,B 0,C 180,E1 29903.487,E2 29903.487} C_VEL
LIN {X 0,Y 619.367,Z 1075.127,A -85,B 0,C 180,E1 29902.946,E2 29902.946} C_VEL
LIN {X 0,Y 618.925,Z 1090.264,A -85,B 0,C 180,E1 29902.212,E2 29902.212} C_VEL
LIN {X 0,Y 618.489,Z 1103.673,A -85,B 0,C 180,E1 29901.383,E2 29901.383} C_VEL
LIN {X 0,Y 618.013,Z 1116.859,A -85,B 0,C 180,E1 29900.356,E2 29900.356} C_VEL
LIN {X 0,Y 617.601,Z 1127.998,A -85,B 0,C 180,E1 29899.286,E2 29899.286} C_VEL
LIN {X 0,Y 617.197,Z 1138.507,A -85,B 0,C 180,E1 29898.023,E2 29898.023} C_VEL
LIN {X 0,Y 616.887,Z 1147.452,A -85,B 0,C 180,E1 29896.672,E2 29896.672} C_VEL
LIN {X 0,Y 616.654,Z 1154.735,A -85,B 0,C 180,E1 29895.229,E2 29895.229} C_VEL
LIN {X 0,Y 616.521,Z 1160.306,A -85,B 0,C 180,E1 29893.728,E2 29893.728} C_VEL
LIN {X 0,Y 616.451,Z 1164.022,A -85,B 0,C 180,E1 29892.173,E2 29892.173} C_VEL
LIN {X 0,Y 616.428,Z 1165.941,A -85,B 0,C 180,E1 29890.6,E2 29890.6} C_VEL
LIN {X 0,Y 616.454,Z 1165.932,A -85,B 0,C 180,E1 29889.052,E2 29889.052} C_VEL
LIN {X 0,Y 616.526,Z 1164.245,A -85,B 0,C 180,E1 29887.549,E2 29887.549} C_VEL
LIN {X 0,Y 616.637,Z 1160.78,A -85,B 0,C 180,E1 29886.05,E2 29886.05} C_VEL
LIN {X 0,Y 616.844,Z 1155.432,A -85,B 0,C 180,E1 29884.54,E2 29884.54} C_VEL
LIN {X 0,Y 617.13,Z 1148.664,A -85,B 0,C 180,E1 29883.158,E2 29883.158} C_VEL
LIN {X 0,Y 617.535,Z 1139.776,A -85,B 0,C 180,E1 29881.763,E2 29881.763} C_VEL
LIN {X 0,Y 617.99,Z 1129.992,A -85,B 0,C 180,E1 29880.556,E2 29880.556} C_VEL
LIN {X 0,Y 618.515,Z 1118.303,A -85,B 0,C 180,E1 29879.398,E2 29879.398} C_VEL
LIN {X 0,Y 619.031,Z 1106.095,A -85,B 0,C 180,E1 29878.426,E2 29878.426} C_VEL
LIN {X 0,Y 619.567,Z 1091.474,A -85,B 0,C 180,E1 29877.503,E2 29877.503} C_VEL
LIN {X 0,Y 620.028,Z 1077.317,A -85,B 0,C 180,E1 29876.811,E2 29876.811} C_VEL
LIN {X 0,Y 620.401,Z 1060.887,A -85,B 0,C 180,E1 29876.211,E2 29876.211} C_VEL
LIN {X 0,Y 620.612,Z 1044.987,A -85,B 0,C 180,E1 29875.816,E2 29875.816} C_VEL
LIN {X 0,Y 624.099,Z 906.452,A -85,B 0,C 180,E1 29873.538,E2 29873.538} C_VEL
LIN {X 0,Y 626.843,Z 861.689,A -85,B 0,C 180,E1 29870.126,E2 29870.126} C_VEL
LIN {X 0,Y 630.128,Z 817.919,A -85,B 0,C 180,E1 29866.698,E2 29866.698} C_VEL
LIN {X 0,Y 634.173,Z 775.544,A -85,B 0,C 180,E1 29863.277,E2 29863.277} C_VEL
LIN {X 0,Y 638.756,Z 736.331,A -85,B 0,C 180,E1 29859.999,E2 29859.999} C_VEL
LIN {X 0,Y 641.835,Z 710.161,A -85,B 0,C 180,E1 29857.659,E2 29857.659} C_VEL
LIN {X 0,Y 637.36,Z 697.825,A -85,B 0,C 180,E1 29855.704,E2 29855.704} C_VEL
LIN {X 0,Y 633.432,Z 688.038,A -85,B 0,C 180,E1 29853.87,E2 29853.87} C_VEL
LIN {X 0,Y 629.994,Z 680.26,A -85,B 0,C 180,E1 29852.082,E2 29852.082} C_VEL
LIN {X 0,Y 627.879,Z 675.89,A -85,B 0,C 180,E1 29850.836,E2 29850.836} C_VEL
LIN {X 0,Y 625.808,Z 671.492,A -85,B 0,C 180,E1 29849.25,E2 29849.25} C_VEL
LIN {X 0,Y 623.96,Z 668.318,A -85,B 0,C 180,E1 29847.275,E2 29847.275} C_VEL
LIN {X 0,Y 623.72,Z 666.954,A -85,B 0,C 180,E1 29845.973,E2 29845.973} C_VEL
LIN {X 0,Y 623.918,Z 667.292,A -85,B 0,C 180,E1 29844.314,E2 29844.314} C_VEL
LIN {X 0,Y 625.099,Z 670.47,A -85,B 0,C 180,E1 29842.335,E2 29842.335} C_VEL
LIN {X 0,Y 626.656,Z 672.248,A -85,B 0,C 180,E1 29841.4,E2 29841.4} C_VEL
LIN {X 0,Y 628.192,Z 675.884,A -85,B 0,C 180,E1 29840.337,E2 29840.337} C_VEL
LIN {X 0,Y 629.24,Z 677.726,A -85,B 0,C 180,E1 29839.823,E2 29839.823} C_VEL
LIN {X 0,Y 631.642,Z 682.745,A -85,B 0,C 180,E1 29838.691,E2 29838.691} C_VEL
LIN {X 0,Y 634.73,Z 689.238,A -85,B 0,C 180,E1 29837.483,E2 29837.483} C_VEL
LIN {X 0,Y 638.839,Z 699.372,A -85,B 0,C 180,E1 29835.978,E2 29835.978} C_VEL
LIN {X 0,Y 640.142,Z 703.537,A -85,B 0,C 180,E1 29835.466,E2 29835.466} C_VEL
LIN {X 0,Y 635.091,Z 742.173,A -85,B 0,C 180,E1 29832.92,E2 29832.92} C_VEL
LIN {X 0,Y 631.708,Z 781.886,A -85,B 0,C 180,E1 29830.417,E2 29830.417} C_VEL
LIN {X 0,Y 632.097,Z 803.066,A -85,B 0,C 180,E1 29829.017,E2 29829.017} C_VEL
LIN {X 0,Y 634.171,Z 818.945,A -85,B 0,C 180,E1 29827.902,E2 29827.902} C_VEL
LIN {X 0,Y 638.063,Z 833.797,A -85,B 0,C 180,E1 29826.796,E2 29826.796} C_VEL
LIN {X 0,Y 643.95,Z 847.58,A -85,B 0,C 180,E1 29825.699,E2 29825.699} C_VEL
LIN {X 0,Y 651.023,Z 858.984,A -85,B 0,C 180,E1 29824.735,E2 29824.735} C_VEL
LIN {X 0,Y 658.877,Z 868.429,A -85,B 0,C 180,E1 29823.89,E2 29823.89} C_VEL
LIN {X 0,Y 668.957,Z 877.653,A -85,B 0,C 180,E1 29823.015,E2 29823.015} C_VEL
LIN {X 0,Y 680.615,Z 885.655,A -85,B 0,C 180,E1 29822.199,E2 29822.199} C_VEL
LIN {X 0,Y 693.17,Z 892.321,A -85,B 0,C 180,E1 29821.46,E2 29821.46} C_VEL
LIN {X 0,Y 663.521,Z 934.885,A -85,B 0,C 180,E1 29820.318,E2 29820.318} C_VEL
LIN {X 0,Y 652.262,Z 953.702,A -85,B 0,C 180,E1 29819.728,E2 29819.728} C_VEL
LIN {X 0,Y 644.512,Z 969.789,A -85,B 0,C 180,E1 29819.151,E2 29819.151} C_VEL
LIN {X 0,Y 640.553,Z 979.287,A -85,B 0,C 180,E1 29818.786,E2 29818.786} C_VEL
LIN {X 0,Y 634.262,Z 993.883,A -85,B 0,C 180,E1 29818.223,E2 29818.223} C_VEL
LIN {X 0,Y 628.198,Z 1013.381,A -85,B 0,C 180,E1 29817.414,E2 29817.414} C_VEL
LIN {X 0,Y 627.25,Z 1029.163,A -85,B 0,C 180,E1 29817.25,E2 29817.25} C_VEL
LIN {X 0,Y 626.712,Z 1064.964,A -85,B 0,C 180,E1 29816.769,E2 29816.769} C_VEL
LIN {X 0,Y 626.049,Z 1086.626,A -85,B 0,C 180,E1 29816.32,E2 29816.32} C_VEL
LIN {X 0,Y 625.235,Z 1108.048,A -85,B 0,C 180,E1 29815.706,E2 29815.706} C_VEL
LIN {X 0,Y 624.238,Z 1129.731,A -85,B 0,C 180,E1 29814.913,E2 29814.913} C_VEL
LIN {X 0,Y 623.251,Z 1149.708,A -85,B 0,C 180,E1 29814.011,E2 29814.011} C_VEL
LIN {X 0,Y 622.111,Z 1170.171,A -85,B 0,C 180,E1 29812.888,E2 29812.888} C_VEL
LIN {X 0,Y 621.013,Z 1189.337,A -85,B 0,C 180,E1 29811.634,E2 29811.634} C_VEL
LIN {X 0,Y 619.927,Z 1207.45,A -85,B 0,C 180,E1 29810.239,E2 29810.239} C_VEL
LIN {X 0,Y 618.843,Z 1227.008,A -85,B 0,C 180,E1 29808.461,E2 29808.461} C_VEL
LIN {X 0,Y 618.214,Z 1239.113,A -85,B 0,C 180,E1 29807.215,E2 29807.215} C_VEL
LIN {X 0,Y 617.621,Z 1251.394,A -85,B 0,C 180,E1 29805.781,E2 29805.781} C_VEL
LIN {X 0,Y 616.996,Z 1265.259,A -85,B 0,C 180,E1 29803.876,E2 29803.876} C_VEL
LIN {X 0,Y 616.637,Z 1274.605,A -85,B 0,C 180,E1 29802.358,E2 29802.358} C_VEL
LIN {X 0,Y 616.366,Z 1282.149,A -85,B 0,C 180,E1 29800.94,E2 29800.94} C_VEL
LIN {X 0,Y 616.173,Z 1288.997,A -85,B 0,C 180,E1 29799.432,E2 29799.432} C_VEL
LIN {X 0,Y 616.041,Z 1294.667,A -85,B 0,C 180,E1 29797.929,E2 29797.929} C_VEL
LIN {X 0,Y 615.962,Z 1299.631,A -85,B 0,C 180,E1 29796.243,E2 29796.243} C_VEL
LIN {X 0,Y 615.918,Z 1304.094,A -85,B 0,C 180,E1 29794.095,E2 29794.095} C_VEL
LIN {X 0,Y 615.907,Z 1306.33,A -85,B 0,C 180,E1 29792.325,E2 29792.325} C_VEL
LIN {X 0,Y 615.905,Z 1307.319,A -85,B 0,C 180,E1 29790.65,E2 29790.65} C_VEL
LIN {X 0,Y 615.913,Z 1307.179,A -85,B 0,C 180,E1 29788.883,E2 29788.883} C_VEL
LIN {X 0,Y 615.919,Z 1305.194,A -85,B 0,C 180,E1 29786.648,E2 29786.648} C_VEL
LIN {X 0,Y 615.933,Z 1302.161,A -85,B 0,C 180,E1 29784.876,E2 29784.876} C_VEL
LIN {X 0,Y 615.976,Z 1298.107,A -85,B 0,C 180,E1 29783.193,E2 29783.193} C_VEL
LIN {X 0,Y 616.084,Z 1293.035,A -85,B 0,C 180,E1 29781.6,E2 29781.6} C_VEL
LIN {X 0,Y 616.291,Z 1284.517,A -85,B 0,C 180,E1 29779.529,E2 29779.529} C_VEL
LIN {X 0,Y 616.593,Z 1275.819,A -85,B 0,C 180,E1 29777.829,E2 29777.829} C_VEL
LIN {X 0,Y 616.945,Z 1266.743,A -85,B 0,C 180,E1 29776.312,E2 29776.312} C_VEL
LIN {X 0,Y 617.498,Z 1254.859,A -85,B 0,C 180,E1 29774.599,E2 29774.599} C_VEL
LIN {X 0,Y 618.191,Z 1240.702,A -85,B 0,C 180,E1 29772.879,E2 29772.879} C_VEL
LIN {X 0,Y 618.904,Z 1227.656,A -85,B 0,C 180,E1 29771.505,E2 29771.505} C_VEL
LIN {X 0,Y 619.722,Z 1213.134,A -85,B 0,C 180,E1 29770.161,E2 29770.161} C_VEL
LIN {X 0,Y 620.813,Z 1194.129,A -85,B 0,C 180,E1 29768.653,E2 29768.653} C_VEL
LIN {X 0,Y 621.889,Z 1175.651,A -85,B 0,C 180,E1 29767.401,E2 29767.401} C_VEL
LIN {X 0,Y 622.966,Z 1155.815,A -85,B 0,C 180,E1 29766.275,E2 29766.275} C_VEL
LIN {X 0,Y 624.049,Z 1134.912,A -85,B 0,C 180,E1 29765.279,E2 29765.279} C_VEL
LIN {X 0,Y 625.024,Z 1114.501,A -85,B 0,C 180,E1 29764.479,E2 29764.479} C_VEL
LIN {X 0,Y 625.905,Z 1092.907,A -85,B 0,C 180,E1 29763.815,E2 29763.815} C_VEL
LIN {X 0,Y 626.666,Z 1070.422,A -85,B 0,C 180,E1 29763.291,E2 29763.291} C_VEL
LIN {X 0,Y 627.208,Z 1048.377,A -85,B 0,C 180,E1 29762.939,E2 29762.939} C_VEL
LIN {X 0,Y 627.845,Z 1019.407,A -85,B 0,C 180,E1 29762.589,E2 29762.589} C_VEL
LIN {X 0,Y 631.971,Z 1005.315,A -85,B 0,C 180,E1 29761.971,E2 29761.971} C_VEL
LIN {X 0,Y 637.125,Z 990.414,A -85,B 0,C 180,E1 29761.35,E2 29761.35} C_VEL
LIN {X 0,Y 643.78,Z 975.452,A -85,B 0,C 180,E1 29760.795,E2 29760.795} C_VEL
LIN {X 0,Y 650.566,Z 960.165,A -85,B 0,C 180,E1 29760.235,E2 29760.235} C_VEL
LIN {X 0,Y 660.503,Z 942.342,A -85,B 0,C 180,E1 29759.677,E2 29759.677} C_VEL
LIN {X 0,Y 676.987,Z 917.154,A -85,B 0,C 180,E1 29759.02,E2 29759.02} C_VEL
LIN {X 0,Y 693.644,Z 892.692,A -85,B 0,C 180,E1 29758.442,E2 29758.442} C_VEL
LIN {X 0,Y 681.764,Z 886.999,A -85,B 0,C 180,E1 29757.648,E2 29757.648} C_VEL
LIN {X 0,Y 670.62,Z 879.615,A -85,B 0,C 180,E1 29756.767,E2 29756.767} C_VEL
LIN {X 0,Y 660.944,Z 870.904,A -85,B 0,C 180,E1 29755.845,E2 29755.845} C_VEL
LIN {X 0,Y 652.733,Z 860.941,A -85,B 0,C 180,E1 29754.886,E2 29754.886} C_VEL
LIN {X 0,Y 645.972,Z 849.708,A -85,B 0,C 180,E1 29753.901,E2 29753.901} C_VEL
LIN {X 0,Y 640.277,Z 835.888,A -85,B 0,C 180,E1 29752.792,E2 29752.792} C_VEL
LIN {X 0,Y 636.493,Z 820.957,A -85,B 0,C 180,E1 29751.692,E2 29751.692} C_VEL
LIN {X 0,Y 634.394,Z 804.312,A -85,B 0,C 180,E1 29750.562,E2 29750.562} C_VEL
LIN {X 0,Y 633.905,Z 783.153,A -85,B 0,C 180,E1 29749.229,E2 29749.229} C_VEL
LIN {X 0,Y 637.201,Z 725.275,A -85,B 0,C 180,E1 29745.772,E2 29745.772} C_VEL
LIN {X 0,Y 638.401,Z 703.494,A -85,B 0,C 180,E1 29744.436,E2 29744.436} C_VEL
LIN {X 0,Y 626.872,Z 677.761,A -85,B 0,C 180,E1 29741.815,E2 29741.815} C_VEL
LIN {X 0,Y 618.383,Z 659.404,A -85,B 0,C 180,E1 29739.815,E2 29739.815} C_VEL
LIN {X 0,Y 617.019,Z 655.81,A -85,B 0,C 180,E1 29739.407,E2 29739.407} C_VEL
LIN {X 0,Y 617.014,Z 655.892,A -85,B 0,C 180,E1 29736.662,E2 29736.662} C_VEL
LIN {X 0,Y 618.41,Z 659.45,A -85,B 0,C 180,E1 29736.213,E2 29736.213} C_VEL
LIN {X 0,Y 622.898,Z 670.344,A -85,B 0,C 180,E1 29734.852,E2 29734.852} C_VEL
LIN {X 0,Y 627.152,Z 683.757,A -85,B 0,C 180,E1 29733.338,E2 29733.338} C_VEL
LIN {X 0,Y 628.929,Z 690.94,A -85,B 0,C 180,E1 29732.582,E2 29732.582} C_VEL
LIN {X 0,Y 628.457,Z 707.224,A -85,B 0,C 180,E1 29731.24,E2 29731.24} C_VEL
LIN {X 0,Y 632.635,Z 726.914,A -85,B 0,C 180,E1 29730.621,E2 29730.621} C_VEL
LIN {X 0,Y 629.458,Z 850.279,A -85,B 0,C 180,E1 29728.844,E2 29728.844} C_VEL
LIN {X 0,Y 627.477,Z 975.525,A -85,B 0,C 180,E1 29727.201,E2 29727.201} C_VEL
LIN {X 0,Y 626.963,Z 1010.786,A -85,B 0,C 180,E1 29726.727,E2 29726.727} C_VEL
LIN {X 0,Y 626.376,Z 1033.011,A -85,B 0,C 180,E1 29726.256,E2 29726.256} C_VEL
LIN {X 0,Y 625.634,Z 1054.405,A -85,B 0,C 180,E1 29725.64,E2 29725.64} C_VEL
LIN {X 0,Y 624.783,Z 1074.857,A -85,B 0,C 180,E1 29724.892,E2 29724.892} C_VEL
LIN {X 0,Y 623.812,Z 1094.882,A -85,B 0,C 180,E1 29723.986,E2 29723.986} C_VEL
LIN {X 0,Y 622.771,Z 1113.585,A -85,B 0,C 180,E1 29722.964,E2 29722.964} C_VEL
LIN {X 0,Y 621.637,Z 1132.871,A -85,B 0,C 180,E1 29721.713,E2 29721.713} C_VEL
LIN {X 0,Y 620.591,Z 1149.885,A -85,B 0,C 180,E1 29720.415,E2 29720.415} C_VEL
LIN {X 0,Y 619.592,Z 1165.367,A -85,B 0,C 180,E1 29719.025,E2 29719.025} C_VEL
LIN {X 0,Y 618.675,Z 1180.023,A -85,B 0,C 180,E1 29717.494,E2 29717.494} C_VEL
LIN {X 0,Y 617.88,Z 1193.393,A -85,B 0,C 180,E1 29715.872,E2 29715.872} C_VEL
LIN {X 0,Y 617.214,Z 1205.314,A -85,B 0,C 180,E1 29714.159,E2 29714.159} C_VEL
LIN {X 0,Y 616.698,Z 1215.879,A -85,B 0,C 180,E1 29712.358,E2 29712.358} C_VEL
LIN {X 0,Y 616.344,Z 1225.117,A -85,B 0,C 180,E1 29710.469,E2 29710.469} C_VEL
LIN {X 0,Y 616.104,Z 1232.538,A -85,B 0,C 180,E1 29708.587,E2 29708.587} C_VEL
LIN {X 0,Y 615.978,Z 1238.562,A -85,B 0,C 180,E1 29706.618,E2 29706.618} C_VEL
LIN {X 0,Y 615.929,Z 1243.222,A -85,B 0,C 180,E1 29704.562,E2 29704.562} C_VEL
LIN {X 0,Y 615.909,Z 1246.065,A -85,B 0,C 180,E1 29702.605,E2 29702.605} C_VEL
LIN {X 0,Y 615.913,Z 1247.36,A -85,B 0,C 180,E1 29700.558,E2 29700.558} C_VEL
LIN {X 0,Y 615.903,Z 1247.117,A -85,B 0,C 180,E1 29698.605,E2 29698.605} C_VEL
LIN {X 0,Y 615.904,Z 1245.273,A -85,B 0,C 180,E1 29696.649,E2 29696.649} C_VEL
LIN {X 0,Y 615.941,Z 1241.704,A -85,B 0,C 180,E1 29694.597,E2 29694.597} C_VEL
LIN {X 0,Y 616.02,Z 1236.474,A -85,B 0,C 180,E1 29692.539,E2 29692.539} C_VEL
LIN {X 0,Y 616.177,Z 1229.919,A -85,B 0,C 180,E1 29690.619,E2 29690.619} C_VEL
LIN {X 0,Y 616.465,Z 1221.551,A -85,B 0,C 180,E1 29688.682,E2 29688.682} C_VEL
LIN {X 0,Y 616.887,Z 1211.576,A -85,B 0,C 180,E1 29686.789,E2 29686.789} C_VEL
LIN {X 0,Y 617.485,Z 1200.176,A -85,B 0,C 180,E1 29684.984,E2 29684.984} C_VEL
LIN {X 0,Y 618.232,Z 1187.257,A -85,B 0,C 180,E1 29683.268,E2 29683.268} C_VEL
LIN {X 0,Y 619.122,Z 1172.965,A -85,B 0,C 180,E1 29681.643,E2 29681.643} C_VEL
LIN {X 0,Y 620.109,Z 1158.01,A -85,B 0,C 180,E1 29680.176,E2 29680.176} C_VEL
LIN {X 0,Y 621.227,Z 1141.136,A -85,B 0,C 180,E1 29678.768,E2 29678.768} C_VEL
LIN {X 0,Y 622.382,Z 1123.141,A -85,B 0,C 180,E1 29677.484,E2 29677.484} C_VEL
LIN {X 0,Y 623.591,Z 1103.776,A -85,B 0,C 180,E1 29676.313,E2 29676.313} C_VEL
LIN {X 0,Y 624.725,Z 1083.963,A -85,B 0,C 180,E1 29675.308,E2 29675.308} C_VEL
LIN {X 0,Y 625.727,Z 1064.135,A -85,B 0,C 180,E1 29674.491,E2 29674.491} C_VEL
LIN {X 0,Y 626.666,Z 1041.935,A -85,B 0,C 180,E1 29673.757,E2 29673.757} C_VEL
LIN {X 0,Y 627.43,Z 1020.335,A -85,B 0,C 180,E1 29673.215,E2 29673.215} C_VEL
LIN {X 0,Y 627.963,Z 998.32,A -85,B 0,C 180,E1 29672.83,E2 29672.83} C_VEL
LIN {X 0,Y 631.283,Z 774.571,A -85,B 0,C 180,E1 29669.989,E2 29669.989} C_VEL
LIN {X 0,Y 630.547,Z 767.003,A -85,B 0,C 180,E1 29669.845,E2 29669.845} C_VEL
LIN {X 0,Y 625.476,Z 747.245,A -85,B 0,C 180,E1 29669.302,E2 29669.302} C_VEL
LIN {X 0,Y 624.946,Z 740.739,A -85,B 0,C 180,E1 29669.181,E2 29669.181} C_VEL
LIN {X 0,Y 624.988,Z 726.947,A -85,B 0,C 180,E1 29668.986,E2 29668.986} C_VEL
LIN {X 0,Y 619.465,Z 702.324,A -85,B 0,C 180,E1 29668.305,E2 29668.305} C_VEL
LIN {X 0,Y 619.885,Z 690.703,A -85,B 0,C 180,E1 29667.291,E2 29667.291} C_VEL
LIN {X 0,Y 613.53,Z 670.239,A -85,B 0,C 180,E1 29665.061,E2 29665.061} C_VEL
LIN {X 0,Y 609.058,Z 656.8,A -85,B 0,C 180,E1 29663.537,E2 29663.537} C_VEL
LIN {X 0,Y 609.074,Z 656.799,A -85,B 0,C 180,E1 29660.312,E2 29660.312} C_VEL
LIN {X 0,Y 609.06,Z 656.802,A -85,B 0,C 180,E1 29657.183,E2 29657.183} C_VEL
LIN {X 0,Y 609.061,Z 656.8,A -85,B 0,C 180,E1 29654.023,E2 29654.023} C_VEL
LIN {X 0,Y 609.065,Z 656.8,A -85,B 0,C 180,E1 29650.798,E2 29650.798} C_VEL
LIN {X 0,Y 609.078,Z 656.795,A -85,B 0,C 180,E1 29647.522,E2 29647.522} C_VEL
LIN {X 0,Y 609.074,Z 656.798,A -85,B 0,C 180,E1 29644.271,E2 29644.271} C_VEL
LIN {X 0,Y 609.081,Z 656.797,A -85,B 0,C 180,E1 29641.025,E2 29641.025} C_VEL
LIN {X 0,Y 609.061,Z 656.797,A -85,B 0,C 180,E1 29637.764,E2 29637.764} C_VEL
LIN {X 0,Y 609.06,Z 656.798,A -85,B 0,C 180,E1 29634.563,E2 29634.563} C_VEL
LIN {X 0,Y 609.059,Z 656.8,A -85,B 0,C 180,E1 29631.433,E2 29631.433} C_VEL
LIN {X 0,Y 609.074,Z 656.803,A -85,B 0,C 180,E1 29628.275,E2 29628.275} C_VEL
LIN {X 0,Y 609.058,Z 656.8,A -85,B 0,C 180,E1 29625.132,E2 29625.132} C_VEL
LIN {X 0,Y 609.058,Z 656.795,A -85,B 0,C 180,E1 29622.035,E2 29622.035} C_VEL
LIN {X 0,Y 609.056,Z 656.793,A -85,B 0,C 180,E1 29618.879,E2 29618.879} C_VEL
LIN {X 0,Y 609.07,Z 656.802,A -85,B 0,C 180,E1 29615.749,E2 29615.749} C_VEL
LIN {X 0,Y 609.059,Z 656.799,A -85,B 0,C 180,E1 29612.542,E2 29612.542} C_VEL
LIN {X 0,Y 609.057,Z 656.793,A -85,B 0,C 180,E1 29609.437,E2 29609.437} C_VEL
LIN {X 0,Y 609.056,Z 656.794,A -85,B 0,C 180,E1 29606.33,E2 29606.33} C_VEL
LIN {X 0,Y 609.061,Z 656.8,A -85,B 0,C 180,E1 29603.213,E2 29603.213} C_VEL
LIN {X 0,Y 609.061,Z 656.802,A -85,B 0,C 180,E1 29600.071,E2 29600.071} C_VEL
LIN {X 0,Y 609.058,Z 656.799,A -85,B 0,C 180,E1 29596.907,E2 29596.907} C_VEL
LIN {X 0,Y 609.057,Z 656.799,A -85,B 0,C 180,E1 29593.796,E2 29593.796} C_VEL
LIN {X 0,Y 609.064,Z 656.8,A -85,B 0,C 180,E1 29590.635,E2 29590.635} C_VEL
LIN {X 0,Y 609.058,Z 656.803,A -85,B 0,C 180,E1 29587.512,E2 29587.512} C_VEL
LIN {X 0,Y 609.061,Z 656.797,A -85,B 0,C 180,E1 29584.318,E2 29584.318} C_VEL
LIN {X 0,Y 609.063,Z 656.798,A -85,B 0,C 180,E1 29581.143,E2 29581.143} C_VEL
LIN {X 0,Y 609.068,Z 656.789,A -85,B 0,C 180,E1 29577.898,E2 29577.898} C_VEL
LIN {X 0,Y 609.075,Z 656.792,A -85,B 0,C 180,E1 29574.587,E2 29574.587} C_VEL
LIN {X 0,Y 609.079,Z 656.795,A -85,B 0,C 180,E1 29571.391,E2 29571.391} C_VEL
LIN {X 0,Y 609.077,Z 656.792,A -85,B 0,C 180,E1 29568.186,E2 29568.186} C_VEL
LIN {X 0,Y 609.084,Z 656.898,A -85,B 0,C 180,E1 29565.345,E2 29565.345} C_VEL
LIN {X 0,Y 618.654,Z 683.489,A -85,B 0,C 180,E1 29562.5,E2 29562.5} C_VEL
LIN {X 0,Y 622.535,Z 695.28,A -85,B 0,C 180,E1 29561.31,E2 29561.31} C_VEL
LIN {X 0,Y 620.665,Z 732.752,A -85,B 0,C 180,E1 29558.451,E2 29558.451} C_VEL
LIN {X 0,Y 618.509,Z 775.43,A -85,B 0,C 180,E1 29555.249,E2 29555.249} C_VEL
LIN {X 0,Y 616.513,Z 819.644,A -85,B 0,C 180,E1 29551.985,E2 29551.985} C_VEL
LIN {X 0,Y 614.573,Z 867.866,A -85,B 0,C 180,E1 29548.47,E2 29548.47} C_VEL
LIN {X 0,Y 613.54,Z 899.705,A -85,B 0,C 180,E1 29546.203,E2 29546.203} C_VEL
LIN {X 0,Y 614.302,Z 907.691,A -85,B 0,C 180,E1 29546.061,E2 29546.061} C_VEL
LIN {X 0,Y 612.232,Z 1043.702,A -85,B 0,C 180,E1 29544.104,E2 29544.104} C_VEL
LIN {X 0,Y 611.977,Z 1060.749,A -85,B 0,C 180,E1 29543.674,E2 29543.674} C_VEL
LIN {X 0,Y 611.608,Z 1076.228,A -85,B 0,C 180,E1 29543.102,E2 29543.102} C_VEL
LIN {X 0,Y 611.143,Z 1091.305,A -85,B 0,C 180,E1 29542.358,E2 29542.358} C_VEL
LIN {X 0,Y 610.681,Z 1104.687,A -85,B 0,C 180,E1 29541.516,E2 29541.516} C_VEL
LIN {X 0,Y 610.18,Z 1117.806,A -85,B 0,C 180,E1 29540.479,E2 29540.479} C_VEL
LIN {X 0,Y 609.725,Z 1129.383,A -85,B 0,C 180,E1 29539.345,E2 29539.345} C_VEL
LIN {X 0,Y 609.3,Z 1139.776,A -85,B 0,C 180,E1 29538.069,E2 29538.069} C_VEL
LIN {X 0,Y 608.971,Z 1148.655,A -85,B 0,C 180,E1 29536.699,E2 29536.699} C_VEL
LIN {X 0,Y 608.723,Z 1155.869,A -85,B 0,C 180,E1 29535.237,E2 29535.237} C_VEL
LIN {X 0,Y 608.585,Z 1161.184,A -85,B 0,C 180,E1 29533.782,E2 29533.782} C_VEL
LIN {X 0,Y 608.51,Z 1164.879,A -85,B 0,C 180,E1 29532.238,E2 29532.238} C_VEL
LIN {X 0,Y 608.485,Z 1166.816,A -85,B 0,C 180,E1 29530.697,E2 29530.697} C_VEL
LIN {X 0,Y 608.508,Z 1166.984,A -85,B 0,C 180,E1 29529.171,E2 29529.171} C_VEL
LIN {X 0,Y 608.593,Z 1165.304,A -85,B 0,C 180,E1 29527.553,E2 29527.553} C_VEL
LIN {X 0,Y 608.72,Z 1161.926,A -85,B 0,C 180,E1 29526.035,E2 29526.035} C_VEL
LIN {X 0,Y 608.939,Z 1156.712,A -85,B 0,C 180,E1 29524.521,E2 29524.521} C_VEL
LIN {X 0,Y 609.255,Z 1149.98,A -85,B 0,C 180,E1 29523.105,E2 29523.105} C_VEL
LIN {X 0,Y 609.689,Z 1141.181,A -85,B 0,C 180,E1 29521.692,E2 29521.692} C_VEL
LIN {X 0,Y 610.179,Z 1131.533,A -85,B 0,C 180,E1 29520.469,E2 29520.469} C_VEL
LIN {X 0,Y 610.762,Z 1119.471,A -85,B 0,C 180,E1 29519.25,E2 29519.25} C_VEL
LIN {X 0,Y 611.342,Z 1106.687,A -85,B 0,C 180,E1 29518.219,E2 29518.219} C_VEL
LIN {X 0,Y 611.895,Z 1092.873,A -85,B 0,C 180,E1 29517.331,E2 29517.331} C_VEL
LIN {X 0,Y 612.396,Z 1078.964,A -85,B 0,C 180,E1 29516.63,E2 29516.63} C_VEL
LIN {X 0,Y 612.794,Z 1062.869,A -85,B 0,C 180,E1 29516.024,E2 29516.024} C_VEL
LIN {X 0,Y 613.034,Z 1047.171,A -85,B 0,C 180,E1 29515.612,E2 29515.612} C_VEL
LIN {X 0,Y 616.928,Z 907.441,A -85,B 0,C 180,E1 29513.205,E2 29513.205} C_VEL
LIN {X 0,Y 619.949,Z 861.911,A -85,B 0,C 180,E1 29509.687,E2 29509.687} C_VEL
LIN {X 0,Y 623.449,Z 818.917,A -85,B 0,C 180,E1 29506.269,E2 29506.269} C_VEL
LIN {X 0,Y 627.651,Z 777.744,A -85,B 0,C 180,E1 29502.902,E2 29502.902} C_VEL
LIN {X 0,Y 632.489,Z 739.415,A -85,B 0,C 180,E1 29499.647,E2 29499.647} C_VEL
LIN {X 0,Y 635.665,Z 714.514,A -85,B 0,C 180,E1 29497.386,E2 29497.386} C_VEL
LIN {X 0,Y 631.555,Z 702.881,A -85,B 0,C 180,E1 29495.493,E2 29495.493} C_VEL
LIN {X 0,Y 627.926,Z 693.584,A -85,B 0,C 180,E1 29493.697,E2 29493.697} C_VEL
LIN {X 0,Y 624.947,Z 686.434,A -85,B 0,C 180,E1 29492.024,E2 29492.024} C_VEL
LIN {X 0,Y 622.794,Z 681.938,A -85,B 0,C 180,E1 29490.681,E2 29490.681} C_VEL
LIN {X 0,Y 621.03,Z 677.892,A -85,B 0,C 180,E1 29489.203,E2 29489.203} C_VEL
LIN {X 0,Y 619.3,Z 674.631,A -85,B 0,C 180,E1 29487.09,E2 29487.09} C_VEL
LIN {X 0,Y 619.183,Z 673.544,A -85,B 0,C 180,E1 29485.919,E2 29485.919} C_VEL
LIN {X 0,Y 619.411,Z 673.961,A -85,B 0,C 180,E1 29484.286,E2 29484.286} C_VEL
LIN {X 0,Y 620.552,Z 677.053,A -85,B 0,C 180,E1 29482.361,E2 29482.361} C_VEL
LIN {X 0,Y 621.989,Z 679.008,A -85,B 0,C 180,E1 29481.41,E2 29481.41} C_VEL
LIN {X 0,Y 623.678,Z 682.573,A -85,B 0,C 180,E1 29480.31,E2 29480.31} C_VEL
LIN {X 0,Y 626.522,Z 688.563,A -85,B 0,C 180,E1 29478.873,E2 29478.873} C_VEL
LIN {X 0,Y 629.486,Z 695.173,A -85,B 0,C 180,E1 29477.611,E2 29477.611} C_VEL
LIN {X 0,Y 633.615,Z 705.747,A -85,B 0,C 180,E1 29476.019,E2 29476.019} C_VEL
LIN {X 0,Y 634.137,Z 707.337,A -85,B 0,C 180,E1 29475.818,E2 29475.818} C_VEL
LIN {X 0,Y 628.513,Z 746.875,A -85,B 0,C 180,E1 29473.161,E2 29473.161} C_VEL
LIN {X 0,Y 625.026,Z 784.454,A -85,B 0,C 180,E1 29470.743,E2 29470.743} C_VEL
LIN {X 0,Y 625.208,Z 805.055,A -85,B 0,C 180,E1 29469.352,E2 29469.352} C_VEL
LIN {X 0,Y 627.132,Z 821.395,A -85,B 0,C 180,E1 29468.183,E2 29468.183} C_VEL
LIN {X 0,Y 630.888,Z 836.561,A -85,B 0,C 180,E1 29467.03,E2 29467.03} C_VEL
LIN {X 0,Y 636.739,Z 850.827,A -85,B 0,C 180,E1 29465.875,E2 29465.875} C_VEL
LIN {X 0,Y 643.9,Z 862.761,A -85,B 0,C 180,E1 29464.85,E2 29464.85} C_VEL
LIN {X 0,Y 652.328,Z 873.128,A -85,B 0,C 180,E1 29463.911,E2 29463.911} C_VEL
LIN {X 0,Y 662.766,Z 882.821,A -85,B 0,C 180,E1 29462.984,E2 29462.984} C_VEL
LIN {X 0,Y 675.159,Z 891.442,A -85,B 0,C 180,E1 29462.1,E2 29462.1} C_VEL
LIN {X 0,Y 682.475,Z 895.676,A -85,B 0,C 180,E1 29461.644,E2 29461.644} C_VEL
LIN {X 0,Y 656.608,Z 932.976,A -85,B 0,C 180,E1 29460.639,E2 29460.639} C_VEL
LIN {X 0,Y 645.198,Z 952.112,A -85,B 0,C 180,E1 29460.036,E2 29460.036} C_VEL
LIN {X 0,Y 637.407,Z 968.293,A -85,B 0,C 180,E1 29459.451,E2 29459.451} C_VEL
LIN {X 0,Y 633.449,Z 977.704,A -85,B 0,C 180,E1 29459.087,E2 29459.087} C_VEL
LIN {X 0,Y 627.122,Z 992.357,A -85,B 0,C 180,E1 29458.522,E2 29458.522} C_VEL
LIN {X 0,Y 621.192,Z 1011.009,A -85,B 0,C 180,E1 29457.746,E2 29457.746} C_VEL
LIN {X 0,Y 619.988,Z 1028.32,A -85,B 0,C 180,E1 29457.568,E2 29457.568} C_VEL
LIN {X 0,Y 619.4,Z 1064.675,A -85,B 0,C 180,E1 29457.073,E2 29457.073} C_VEL
LIN {X 0,Y 618.691,Z 1086.35,A -85,B 0,C 180,E1 29456.617,E2 29456.617} C_VEL
LIN {X 0,Y 617.837,Z 1107.334,A -85,B 0,C 180,E1 29456.011,E2 29456.011} C_VEL
LIN {X 0,Y 616.814,Z 1128.51,A -85,B 0,C 180,E1 29455.234,E2 29455.234} C_VEL
LIN {X 0,Y 615.725,Z 1148.921,A -85,B 0,C 180,E1 29454.308,E2 29454.308} C_VEL
LIN {X 0,Y 614.579,Z 1168.339,A -85,B 0,C 180,E1 29453.235,E2 29453.235} C_VEL
LIN {X 0,Y 613.43,Z 1187.056,A -85,B 0,C 180,E1 29452.016,E2 29452.016} C_VEL
LIN {X 0,Y 612.316,Z 1204.952,A -85,B 0,C 180,E1 29450.652,E2 29450.652} C_VEL
LIN {X 0,Y 611.252,Z 1222.307,A -85,B 0,C 180,E1 29449.095,E2 29449.095} C_VEL
LIN {X 0,Y 610.381,Z 1237.02,A -85,B 0,C 180,E1 29447.541,E2 29447.541} C_VEL
LIN {X 0,Y 609.555,Z 1253.062,A -85,B 0,C 180,E1 29445.604,E2 29445.604} C_VEL
LIN {X 0,Y 608.993,Z 1265.199,A -85,B 0,C 180,E1 29443.868,E2 29443.868} C_VEL
LIN {X 0,Y 608.659,Z 1273.927,A -85,B 0,C 180,E1 29442.426,E2 29442.426} C_VEL
LIN {X 0,Y 608.385,Z 1281.459,A -85,B 0,C 180,E1 29440.989,E2 29440.989} C_VEL
LIN {X 0,Y 608.208,Z 1287.902,A -85,B 0,C 180,E1 29439.556,E2 29439.556} C_VEL
LIN {X 0,Y 608.076,Z 1293.656,A -85,B 0,C 180,E1 29438.033,E2 29438.033} C_VEL
LIN {X 0,Y 607.989,Z 1298.591,A -85,B 0,C 180,E1 29436.42,E2 29436.42} C_VEL
LIN {X 0,Y 607.935,Z 1303.306,A -85,B 0,C 180,E1 29434.338,E2 29434.338} C_VEL
LIN {X 0,Y 607.915,Z 1305.878,A -85,B 0,C 180,E1 29432.45,E2 29432.45} C_VEL
LIN {X 0,Y 607.919,Z 1306.955,A -85,B 0,C 180,E1 29430.847,E2 29430.847} C_VEL
LIN {X 0,Y 607.915,Z 1306.983,A -85,B 0,C 180,E1 29429.245,E2 29429.245} C_VEL
LIN {X 0,Y 607.913,Z 1305.968,A -85,B 0,C 180,E1 29427.642,E2 29427.642} C_VEL
LIN {X 0,Y 607.927,Z 1303.756,A -85,B 0,C 180,E1 29425.943,E2 29425.943} C_VEL
LIN {X 0,Y 607.969,Z 1299.443,A -85,B 0,C 180,E1 29423.862,E2 29423.862} C_VEL
LIN {X 0,Y 608.071,Z 1293.756,A -85,B 0,C 180,E1 29421.964,E2 29421.964} C_VEL
LIN {X 0,Y 608.21,Z 1287.671,A -85,B 0,C 180,E1 29420.346,E2 29420.346} C_VEL
LIN {X 0,Y 608.444,Z 1279.853,A -85,B 0,C 180,E1 29418.625,E2 29418.625} C_VEL
LIN {X 0,Y 608.865,Z 1268.71,A -85,B 0,C 180,E1 29416.61,E2 29416.61} C_VEL
LIN {X 0,Y 609.352,Z 1257.872,A -85,B 0,C 180,E1 29414.973,E2 29414.973} C_VEL
LIN {X 0,Y 609.911,Z 1246.849,A -85,B 0,C 180,E1 29413.523,E2 29413.523} C_VEL
LIN {X 0,Y 610.704,Z 1232.492,A -85,B 0,C 180,E1 29411.875,E2 29411.875} C_VEL
LIN {X 0,Y 611.616,Z 1216.62,A -85,B 0,C 180,E1 29410.334,E2 29410.334} C_VEL
LIN {X 0,Y 612.497,Z 1202.283,A -85,B 0,C 180,E1 29409.114,E2 29409.114} C_VEL
LIN {X 0,Y 613.578,Z 1184.374,A -85,B 0,C 180,E1 29407.785,E2 29407.785} C_VEL
LIN {X 0,Y 614.704,Z 1165.771,A -85,B 0,C 180,E1 29406.615,E2 29406.615} C_VEL
LIN {X 0,Y 615.864,Z 1144.869,A -85,B 0,C 180,E1 29405.507,E2 29405.507} C_VEL
LIN {X 0,Y 616.988,Z 1124.051,A -85,B 0,C 180,E1 29404.592,E2 29404.592} C_VEL
LIN {X 0,Y 617.953,Z 1103.332,A -85,B 0,C 180,E1 29403.862,E2 29403.862} C_VEL
LIN {X 0,Y 618.867,Z 1080.743,A -85,B 0,C 180,E1 29403.245,E2 29403.245} C_VEL
LIN {X 0,Y 619.582,Z 1058.821,A -85,B 0,C 180,E1 29402.808,E2 29402.808} C_VEL
LIN {X 0,Y 620.435,Z 1019.698,A -85,B 0,C 180,E1 29402.309,E2 29402.309} C_VEL
LIN {X 0,Y 621.194,Z 1016.099,A -85,B 0,C 180,E1 29402.173,E2 29402.173} C_VEL
LIN {X 0,Y 628.523,Z 993.182,A -85,B 0,C 180,E1 29401.181,E2 29401.181} C_VEL
LIN {X 0,Y 634.971,Z 978.545,A -85,B 0,C 180,E1 29400.624,E2 29400.624} C_VEL
LIN {X 0,Y 643.317,Z 959.539,A -85,B 0,C 180,E1 29399.916,E2 29399.916} C_VEL
LIN {X 0,Y 653.213,Z 941.621,A -85,B 0,C 180,E1 29399.347,E2 29399.347} C_VEL
LIN {X 0,Y 668.372,Z 918.297,A -85,B 0,C 180,E1 29398.726,E2 29398.726} C_VEL
LIN {X 0,Y 683.295,Z 896.524,A -85,B 0,C 180,E1 29398.21,E2 29398.21} C_VEL
LIN {X 0,Y 671.14,Z 889.667,A -85,B 0,C 180,E1 29397.327,E2 29397.327} C_VEL
LIN {X 0,Y 661.025,Z 882.004,A -85,B 0,C 180,E1 29396.457,E2 29396.457} C_VEL
LIN {X 0,Y 651.626,Z 872.568,A -85,B 0,C 180,E1 29395.488,E2 29395.488} C_VEL
LIN {X 0,Y 643.147,Z 860.878,A -85,B 0,C 180,E1 29394.4,E2 29394.4} C_VEL
LIN {X 0,Y 636.818,Z 848.613,A -85,B 0,C 180,E1 29393.354,E2 29393.354} C_VEL
LIN {X 0,Y 632.016,Z 834.982,A -85,B 0,C 180,E1 29392.283,E2 29392.283} C_VEL
LIN {X 0,Y 628.654,Z 819.003,A -85,B 0,C 180,E1 29391.122,E2 29391.122} C_VEL
LIN {X 0,Y 627.014,Z 799.959,A -85,B 0,C 180,E1 29389.85,E2 29389.85} C_VEL
LIN {X 0,Y 627.29,Z 776.908,A -85,B 0,C 180,E1 29388.419,E2 29388.419} C_VEL
LIN {X 0,Y 630.392,Z 728.208,A -85,B 0,C 180,E1 29385.486,E2 29385.486} C_VEL
LIN {X 0,Y 631.692,Z 707.19,A -85,B 0,C 180,E1 29384.188,E2 29384.188} C_VEL
LIN {X 0,Y 619.717,Z 680.265,A -85,B 0,C 180,E1 29381.416,E2 29381.416} C_VEL
LIN {X 0,Y 610.509,Z 660.456,A -85,B 0,C 180,E1 29379.212,E2 29379.212} C_VEL
LIN {X 0,Y 609.071,Z 656.801,A -85,B 0,C 180,E1 29378.798,E2 29378.798} C_VEL
LIN {X 0,Y 609.077,Z 656.95,A -85,B 0,C 180,E1 29377.417,E2 29377.417} C_VEL
LIN {X 0,Y 610.482,Z 660.435,A -85,B 0,C 180,E1 29376.938,E2 29376.938} C_VEL
LIN {X 0,Y 614.487,Z 669.458,A -85,B 0,C 180,E1 29375.71,E2 29375.71} C_VEL
LIN {X 0,Y 618.932,Z 681.943,A -85,B 0,C 180,E1 29374.193,E2 29374.193} C_VEL
LIN {X 0,Y 622.163,Z 694.124,A -85,B 0,C 180,E1 29372.848,E2 29372.848} C_VEL
LIN {X 0,Y 621.727,Z 708.086,A -85,B 0,C 180,E1 29371.694,E2 29371.694} C_VEL
LIN {X 0,Y 626.025,Z 728.138,A -85,B 0,C 180,E1 29371.021,E2 29371.021} C_VEL
LIN {X 0,Y 622.564,Z 845.011,A -85,B 0,C 180,E1 29369.274,E2 29369.274} C_VEL
LIN {X 0,Y 620.345,Z 963.04,A -85,B 0,C 180,E1 29367.664,E2 29367.664} C_VEL
LIN {X 0,Y 619.626,Z 1009.819,A -85,B 0,C 180,E1 29367.033,E2 29367.033} C_VEL
LIN {X 0,Y 619.01,Z 1031.926,A -85,B 0,C 180,E1 29366.57,E2 29366.57} C_VEL
LIN {X 0,Y 618.204,Z 1054.543,A -85,B 0,C 180,E1 29365.918,E2 29365.918} C_VEL
LIN {X 0,Y 617.307,Z 1075.016,A -85,B 0,C 180,E1 29365.163,E2 29365.163} C_VEL
LIN {X 0,Y 616.269,Z 1095.281,A -85,B 0,C 180,E1 29364.236,E2 29364.236} C_VEL
LIN {X 0,Y 615.138,Z 1114.612,A -85,B 0,C 180,E1 29363.164,E2 29363.164} C_VEL
LIN {X 0,Y 613.95,Z 1133.829,A -85,B 0,C 180,E1 29361.898,E2 29361.898} C_VEL
LIN {X 0,Y 612.85,Z 1150.769,A -85,B 0,C 180,E1 29360.585,E2 29360.585} C_VEL
LIN {X 0,Y 611.788,Z 1166.554,A -85,B 0,C 180,E1 29359.148,E2 29359.148} C_VEL
LIN {X 0,Y 610.845,Z 1180.87,A -85,B 0,C 180,E1 29357.628,E2 29357.628} C_VEL
LIN {X 0,Y 610.009,Z 1194.194,A -85,B 0,C 180,E1 29355.984,E2 29355.984} C_VEL
LIN {X 0,Y 609.31,Z 1206.104,A -85,B 0,C 180,E1 29354.25,E2 29354.25} C_VEL
LIN {X 0,Y 608.764,Z 1216.622,A -85,B 0,C 180,E1 29352.425,E2 29352.425} C_VEL
LIN {X 0,Y 608.387,Z 1225.811,A -85,B 0,C 180,E1 29350.511,E2 29350.511} C_VEL
LIN {X 0,Y 608.126,Z 1233.553,A -85,B 0,C 180,E1 29348.51,E2 29348.51} C_VEL
LIN {X 0,Y 607.996,Z 1239.412,A -85,B 0,C 180,E1 29346.516,E2 29346.516} C_VEL
LIN {X 0,Y 607.936,Z 1243.845,A -85,B 0,C 180,E1 29344.434,E2 29344.434} C_VEL
LIN {X 0,Y 607.91,Z 1246.54,A -85,B 0,C 180,E1 29342.451,E2 29342.451} C_VEL
LIN {X 0,Y 607.91,Z 1247.631,A -85,B 0,C 180,E1 29340.377,E2 29340.377} C_VEL
LIN {X 0,Y 607.917,Z 1247.074,A -85,B 0,C 180,E1 29338.209,E2 29338.209} C_VEL
LIN {X 0,Y 607.92,Z 1245.063,A -85,B 0,C 180,E1 29336.228,E2 29336.228} C_VEL
LIN {X 0,Y 607.961,Z 1241.394,A -85,B 0,C 180,E1 29334.242,E2 29334.242} C_VEL
LIN {X 0,Y 608.058,Z 1235.871,A -85,B 0,C 180,E1 29332.155,E2 29332.155} C_VEL
LIN {X 0,Y 608.259,Z 1228.878,A -85,B 0,C 180,E1 29330.156,E2 29330.156} C_VEL
LIN {X 0,Y 608.595,Z 1220.399,A -85,B 0,C 180,E1 29328.245,E2 29328.245} C_VEL
LIN {X 0,Y 609.062,Z 1210.353,A -85,B 0,C 180,E1 29326.382,E2 29326.382} C_VEL
LIN {X 0,Y 609.707,Z 1198.915,A -85,B 0,C 180,E1 29324.593,E2 29324.593} C_VEL
LIN {X 0,Y 610.529,Z 1185.762,A -85,B 0,C 180,E1 29322.855,E2 29322.855} C_VEL
LIN {X 0,Y 611.5,Z 1171.177,A -85,B 0,C 180,E1 29321.219,E2 29321.219} C_VEL
LIN {X 0,Y 612.671,Z 1154.37,A -85,B 0,C 180,E1 29319.608,E2 29319.608} C_VEL
LIN {X 0,Y 613.831,Z 1137.807,A -85,B 0,C 180,E1 29318.248,E2 29318.248} C_VEL
LIN {X 0,Y 615.074,Z 1119.703,A -85,B 0,C 180,E1 29316.985,E2 29316.985} C_VEL
LIN {X 0,Y 616.274,Z 1100.733,A -85,B 0,C 180,E1 29315.866,E2 29315.866} C_VEL
LIN {X 0,Y 617.509,Z 1079.973,A -85,B 0,C 180,E1 29314.844,E2 29314.844} C_VEL
LIN {X 0,Y 618.579,Z 1059.54,A -85,B 0,C 180,E1 29314.02,E2 29314.02} C_VEL
LIN {X 0,Y 619.52,Z 1037.965,A -85,B 0,C 180,E1 29313.34,E2 29313.34} C_VEL
LIN {X 0,Y 620.238,Z 1016.119,A -85,B 0,C 180,E1 29312.824,E2 29312.824} C_VEL
LIN {X 0,Y 620.811,Z 992.321,A -85,B 0,C 180,E1 29312.44,E2 29312.44} C_VEL
LIN {X 0,Y 624.289,Z 775.468,A -85,B 0,C 180,E1 29309.641,E2 29309.641} C_VEL
LIN {X 0,Y 624.946,Z 740.739,A -85,B 0,C 180,E1 29309.181,E2 29309.181} C_VEL
LIN {X 0,Y 624.169,Z 734.323,A -85,B 0,C 180,E1 29309.047,E2 29309.047} C_VEL
LIN {X 0,Y 621.254,Z 726.412,A -85,B 0,C 180,E1 29308.772,E2 29308.772} C_VEL
LIN {X 0,Y 614.92,Z 712.97,A -85,B 0,C 180,E1 29308.219,E2 29308.219} C_VEL
LIN {X 0,Y 613.662,Z 708.816,A -85,B 0,C 180,E1 29308.086,E2 29308.086} C_VEL
LIN {X 0,Y 612.295,Z 702.447,A -85,B 0,C 180,E1 29307.89,E2 29307.89} C_VEL
LIN {X 0,Y 612.512,Z 693.208,A -85,B 0,C 180,E1 29307.071,E2 29307.071} C_VEL
LIN {X 0,Y 605.811,Z 671.799,A -85,B 0,C 180,E1 29304.713,E2 29304.713} C_VEL
LIN {X 0,Y 601.134,Z 657.791,A -85,B 0,C 180,E1 29303.096,E2 29303.096} C_VEL
LIN {X 0,Y 601.129,Z 657.79,A -85,B 0,C 180,E1 29299.773,E2 29299.773} C_VEL
LIN {X 0,Y 601.129,Z 657.789,A -85,B 0,C 180,E1 29296.609,E2 29296.609} C_VEL
LIN {X 0,Y 601.141,Z 657.793,A -85,B 0,C 180,E1 29293.375,E2 29293.375} C_VEL
LIN {X 0,Y 601.122,Z 657.79,A -85,B 0,C 180,E1 29290.196,E2 29290.196} C_VEL
LIN {X 0,Y 601.12,Z 657.784,A -85,B 0,C 180,E1 29287.02,E2 29287.02} C_VEL
LIN {X 0,Y 601.12,Z 657.788,A -85,B 0,C 180,E1 29283.865,E2 29283.865} C_VEL
LIN {X 0,Y 601.13,Z 657.786,A -85,B 0,C 180,E1 29280.688,E2 29280.688} C_VEL
LIN {X 0,Y 601.119,Z 657.789,A -85,B 0,C 180,E1 29277.544,E2 29277.544} C_VEL
LIN {X 0,Y 601.121,Z 657.787,A -85,B 0,C 180,E1 29274.364,E2 29274.364} C_VEL
LIN {X 0,Y 601.121,Z 657.788,A -85,B 0,C 180,E1 29271.262,E2 29271.262} C_VEL
LIN {X 0,Y 601.13,Z 657.791,A -85,B 0,C 180,E1 29268.123,E2 29268.123} C_VEL
LIN {X 0,Y 601.125,Z 657.792,A -85,B 0,C 180,E1 29264.89,E2 29264.89} C_VEL
LIN {X 0,Y 601.128,Z 657.785,A -85,B 0,C 180,E1 29261.612,E2 29261.612} C_VEL
LIN {X 0,Y 601.136,Z 657.778,A -85,B 0,C 180,E1 29258.235,E2 29258.235} C_VEL
LIN {X 0,Y 601.125,Z 657.784,A -85,B 0,C 180,E1 29254.963,E2 29254.963} C_VEL
LIN {X 0,Y 601.121,Z 657.788,A -85,B 0,C 180,E1 29251.717,E2 29251.717} C_VEL
LIN {X 0,Y 601.137,Z 657.791,A -85,B 0,C 180,E1 29248.524,E2 29248.524} C_VEL
LIN {X 0,Y 601.136,Z 657.785,A -85,B 0,C 180,E1 29245.231,E2 29245.231} C_VEL
LIN {X 0,Y 601.119,Z 657.784,A -85,B 0,C 180,E1 29242.066,E2 29242.066} C_VEL
LIN {X 0,Y 601.121,Z 657.782,A -85,B 0,C 180,E1 29238.876,E2 29238.876} C_VEL
LIN {X 0,Y 601.135,Z 657.784,A -85,B 0,C 180,E1 29235.652,E2 29235.652} C_VEL
LIN {X 0,Y 601.138,Z 657.789,A -85,B 0,C 180,E1 29232.38,E2 29232.38} C_VEL
LIN {X 0,Y 601.136,Z 657.789,A -85,B 0,C 180,E1 29229.15,E2 29229.15} C_VEL
LIN {X 0,Y 601.134,Z 657.789,A -85,B 0,C 180,E1 29225.948,E2 29225.948} C_VEL
LIN {X 0,Y 601.127,Z 657.785,A -85,B 0,C 180,E1 29222.653,E2 29222.653} C_VEL
LIN {X 0,Y 601.123,Z 657.789,A -85,B 0,C 180,E1 29219.5,E2 29219.5} C_VEL
LIN {X 0,Y 601.121,Z 657.795,A -85,B 0,C 180,E1 29216.273,E2 29216.273} C_VEL
LIN {X 0,Y 601.134,Z 657.788,A -85,B 0,C 180,E1 29213.099,E2 29213.099} C_VEL
LIN {X 0,Y 601.124,Z 657.791,A -85,B 0,C 180,E1 29209.921,E2 29209.921} C_VEL
LIN {X 0,Y 601.12,Z 657.792,A -85,B 0,C 180,E1 29206.743,E2 29206.743} C_VEL
LIN {X 0,Y 601.141,Z 657.887,A -85,B 0,C 180,E1 29205.821,E2 29205.821} C_VEL
LIN {X 0,Y 610.77,Z 684.488,A -85,B 0,C 180,E1 29202.925,E2 29202.925} C_VEL
LIN {X 0,Y 615.33,Z 698.556,A -85,B 0,C 180,E1 29201.49,E2 29201.49} C_VEL
LIN {X 0,Y 613.338,Z 736.486,A -85,B 0,C 180,E1 29198.577,E2 29198.577} C_VEL
LIN {X 0,Y 611.104,Z 778.567,A -85,B 0,C 180,E1 29195.396,E2 29195.396} C_VEL
LIN {X 0,Y 609.012,Z 822.255,A -85,B 0,C 180,E1 29192.138,E2 29192.138} C_VEL
LIN {X 0,Y 607.006,Z 869.812,A -85,B 0,C 180,E1 29188.643,E2 29188.643} C_VEL
LIN {X 0,Y 605.951,Z 900.262,A -85,B 0,C 180,E1 29186.454,E2 29186.454} C_VEL
LIN {X 0,Y 606.75,Z 908.576,A -85,B 0,C 180,E1 29186.302,E2 29186.302} C_VEL
LIN {X 0,Y 604.511,Z 1044.469,A -85,B 0,C 180,E1 29184.293,E2 29184.293} C_VEL
LIN {X 0,Y 604.248,Z 1061.121,A -85,B 0,C 180,E1 29183.866,E2 29183.866} C_VEL
LIN {X 0,Y 603.882,Z 1076.138,A -85,B 0,C 180,E1 29183.312,E2 29183.312} C_VEL
LIN {X 0,Y 603.391,Z 1091.369,A -85,B 0,C 180,E1 29182.558,E2 29182.558} C_VEL
LIN {X 0,Y 602.872,Z 1105.601,A -85,B 0,C 180,E1 29181.656,E2 29181.656} C_VEL
LIN {X 0,Y 602.327,Z 1119.061,A -85,B 0,C 180,E1 29180.573,E2 29180.573} C_VEL
LIN {X 0,Y 601.841,Z 1130.7,A -85,B 0,C 180,E1 29179.407,E2 29179.407} C_VEL
LIN {X 0,Y 601.397,Z 1141.018,A -85,B 0,C 180,E1 29178.114,E2 29178.114} C_VEL
LIN {X 0,Y 601.049,Z 1149.814,A -85,B 0,C 180,E1 29176.726,E2 29176.726} C_VEL
LIN {X 0,Y 600.79,Z 1156.981,A -85,B 0,C 180,E1 29175.246,E2 29175.246} C_VEL
LIN {X 0,Y 600.646,Z 1162.252,A -85,B 0,C 180,E1 29173.772,E2 29173.772} C_VEL
LIN {X 0,Y 600.565,Z 1165.9,A -85,B 0,C 180,E1 29172.207,E2 29172.207} C_VEL
LIN {X 0,Y 600.543,Z 1167.811,A -85,B 0,C 180,E1 29170.65,E2 29170.65} C_VEL
LIN {X 0,Y 600.572,Z 1167.927,A -85,B 0,C 180,E1 29169.1,E2 29169.1} C_VEL
LIN {X 0,Y 600.668,Z 1166.228,A -85,B 0,C 180,E1 29167.46,E2 29167.46} C_VEL
LIN {X 0,Y 600.809,Z 1162.793,A -85,B 0,C 180,E1 29165.923,E2 29165.923} C_VEL
LIN {X 0,Y 601.062,Z 1157.557,A -85,B 0,C 180,E1 29164.389,E2 29164.389} C_VEL
LIN {X 0,Y 601.406,Z 1150.767,A -85,B 0,C 180,E1 29162.954,E2 29162.954} C_VEL
LIN {X 0,Y 601.882,Z 1141.946,A -85,B 0,C 180,E1 29161.523,E2 29161.523} C_VEL
LIN {X 0,Y 602.415,Z 1132.261,A -85,B 0,C 180,E1 29160.285,E2 29160.285} C_VEL
LIN {X 0,Y 603.055,Z 1120.214,A -85,B 0,C 180,E1 29159.05,E2 29159.05} C_VEL
LIN {X 0,Y 603.676,Z 1107.377,A -85,B 0,C 180,E1 29158.007,E2 29158.007} C_VEL
LIN {X 0,Y 604.277,Z 1093.564,A -85,B 0,C 180,E1 29157.107,E2 29157.107} C_VEL
LIN {X 0,Y 604.801,Z 1079.534,A -85,B 0,C 180,E1 29156.398,E2 29156.398} C_VEL
LIN {X 0,Y 605.233,Z 1063.459,A -85,B 0,C 180,E1 29155.784,E2 29155.784} C_VEL
LIN {X 0,Y 605.477,Z 1047.536,A -85,B 0,C 180,E1 29155.367,E2 29155.367} C_VEL
LIN {X 0,Y 609.76,Z 908.75,A -85,B 0,C 180,E1 29152.888,E2 29152.888} C_VEL
LIN {X 0,Y 613.052,Z 862.764,A -85,B 0,C 180,E1 29149.284,E2 29149.284} C_VEL
LIN {X 0,Y 616.81,Z 819.926,A -85,B 0,C 180,E1 29145.831,E2 29145.831} C_VEL
LIN {X 0,Y 621.324,Z 779.127,A -85,B 0,C 180,E1 29142.438,E2 29142.438} C_VEL
LIN {X 0,Y 626.348,Z 742.076,A -85,B 0,C 180,E1 29139.243,E2 29139.243} C_VEL
LIN {X 0,Y 629.544,Z 718.839,A -85,B 0,C 180,E1 29137.097,E2 29137.097} C_VEL
LIN {X 0,Y 625.58,Z 707.254,A -85,B 0,C 180,E1 29135.142,E2 29135.142} C_VEL
LIN {X 0,Y 622.392,Z 698.976,A -85,B 0,C 180,E1 29133.473,E2 29133.473} C_VEL
LIN {X 0,Y 619.759,Z 692.399,A -85,B 0,C 180,E1 29131.894,E2 29131.894} C_VEL
LIN {X 0,Y 617.772,Z 688.047,A -85,B 0,C 180,E1 29130.545,E2 29130.545} C_VEL
LIN {X 0,Y 616.246,Z 684.277,A -85,B 0,C 180,E1 29129.125,E2 29129.125} C_VEL
LIN {X 0,Y 614.663,Z 681.054,A -85,B 0,C 180,E1 29126.978,E2 29126.978} C_VEL
LIN {X 0,Y 614.64,Z 680.131,A -85,B 0,C 180,E1 29125.858,E2 29125.858} C_VEL
LIN {X 0,Y 614.874,Z 680.467,A -85,B 0,C 180,E1 29124.395,E2 29124.395} C_VEL
